// TIA Portal V20 export
DATA_BLOCK "CallEquipmentMotionCycle_DB"   // DB191
// stored: AssignedProDiagFB Unit1.Em1.ProDiag, InstanceOfName Unit1.Em1.CallEquipmentMotionCycle, InstanceOfType FB, Namespace Unit1.Em1
"Unit1.Em1.CallEquipmentMotionCycle"
   // VAR_INPUT
   //    diameter : LReal := 0.0;
   //    dancer : LReal := 0.105758101851848;
   // END_VAR
   // VAR_OUTPUT
   //    error { ExternalAccessible := 'False'; ExternalVisible := 'False'; ExternalWritable := 'False'} : Bool := FALSE;
   // END_VAR
   // VAR_IN_OUT
   //    syncNode : "Unit1.Em1.typeSyncNode";
   //    axis : Array[1.._.U1EM1_NO_OF_AXES] of DB_ANY;
   // END_VAR
   // VAR
   //    instSequenceUnwinderCycle : "Unit1.Em1.SequenceUnwinderCycle";
   // END_VAR
BEGIN
   instSequenceUnwinderCycle.enableHpMotion := FALSE;
   instSequenceUnwinderCycle.diameter := 0.0;
   instSequenceUnwinderCycle.dancer := 0.105758101851848;
   instSequenceUnwinderCycle.busy := FALSE;
   instSequenceUnwinderCycle.error := FALSE;
   instSequenceUnwinderCycle.slave := 141;
   instSequenceUnwinderCycle.master := 85;
   instSequenceUnwinderCycle.statFirstCall := FALSE;
   instSequenceUnwinderCycle.statDiameter := 0.0;
   instSequenceUnwinderCycle.statFrictionMeasurement.in.execute := FALSE;
   instSequenceUnwinderCycle.statFrictionMeasurement.in.abort := FALSE;
   instSequenceUnwinderCycle.statFrictionMeasurement.in.warmUpTime := T#30S;
   instSequenceUnwinderCycle.statFrictionMeasurement.in.rampTime := 1000.0;
   instSequenceUnwinderCycle.statFrictionMeasurement.in.noOfMeasurementPoints := 100;
   instSequenceUnwinderCycle.statFrictionMeasurement.in.sizeOfArray := 10;
   instSequenceUnwinderCycle.statFrictionMeasurement.in.maxSpeed := 0.0;
   instSequenceUnwinderCycle.statFrictionMeasurement.in.speedValues.values[0] := 100.0;
   instSequenceUnwinderCycle.statFrictionMeasurement.in.speedValues.values[1] := 200.0;
   instSequenceUnwinderCycle.statFrictionMeasurement.in.speedValues.values[2] := 300.0;
   instSequenceUnwinderCycle.statFrictionMeasurement.in.speedValues.values[3] := 400.0;
   instSequenceUnwinderCycle.statFrictionMeasurement.in.speedValues.values[4] := 500.0;
   instSequenceUnwinderCycle.statFrictionMeasurement.in.speedValues.values[5] := 600.0;
   instSequenceUnwinderCycle.statFrictionMeasurement.in.speedValues.values[6] := 700.0;
   instSequenceUnwinderCycle.statFrictionMeasurement.in.speedValues.values[7] := 800.0;
   instSequenceUnwinderCycle.statFrictionMeasurement.in.speedValues.values[8] := 900.0;
   instSequenceUnwinderCycle.statFrictionMeasurement.in.speedValues.values[9] := 1000.0;
   instSequenceUnwinderCycle.statFrictionMeasurement.in.speedValues.values[10..19] := 0.0;
   instSequenceUnwinderCycle.statFrictionMeasurement.in.measurementDelayTime := T#1S;
   instSequenceUnwinderCycle.statFrictionMeasurement.out.done := FALSE;
   instSequenceUnwinderCycle.statFrictionMeasurement.out.valid := FALSE;
   instSequenceUnwinderCycle.statFrictionMeasurement.out.aborted := FALSE;
   instSequenceUnwinderCycle.statFrictionMeasurement.out.busy := FALSE;
   instSequenceUnwinderCycle.statFrictionMeasurement.out.error := FALSE;
   instSequenceUnwinderCycle.statFrictionMeasurement.out.subfunctionState := 16#0000;
   instSequenceUnwinderCycle.statFrictionMeasurement.out.status := 16#7000;
   instSequenceUnwinderCycle.statMaxAcceleration := 360000.0;
   instSequenceUnwinderCycle.statMaxDeceleration := 360000.0;
   instSequenceUnwinderCycle.statUnitsLengthUnit := 1013;
   instSequenceUnwinderCycle.statUnitsVelocityUnit := 1062;
   instSequenceUnwinderCycle.statMechanicsLeadScrew := 10.0;
   instSequenceUnwinderCycle.statLengthConversion := 0.001;
   instSequenceUnwinderCycle.statVelocityConversion := 0.06;
   instSequenceUnwinderCycle.statAccelerationConversion := 0.001;
   instSequenceUnwinderCycle.instLConSMC_Winder.enable := FALSE;
   instSequenceUnwinderCycle.instLConSMC_Winder.speedMatch := FALSE;
   instSequenceUnwinderCycle.instLConSMC_Winder.cntrlEnable := FALSE;
   instSequenceUnwinderCycle.instLConSMC_Winder.jogPos := FALSE;
   instSequenceUnwinderCycle.instLConSMC_Winder.jogNeg := FALSE;
   instSequenceUnwinderCycle.instLConSMC_Winder.lineAxisMotionVector.s := 0.0;
   instSequenceUnwinderCycle.instLConSMC_Winder.lineAxisMotionVector.v := 0.0;
   instSequenceUnwinderCycle.instLConSMC_Winder.lineAxisMotionVector."a" := 0.0;
   instSequenceUnwinderCycle.instLConSMC_Winder.lineAxisActualValues.s := 0.0;
   instSequenceUnwinderCycle.instLConSMC_Winder.lineAxisActualValues.v := 0.0;
   instSequenceUnwinderCycle.instLConSMC_Winder.additionalVelocity := 0.0;
   instSequenceUnwinderCycle.instLConSMC_Winder.typeOfWinder := 2;
   instSequenceUnwinderCycle.instLConSMC_Winder.controlMode := 0;
   instSequenceUnwinderCycle.instLConSMC_Winder.typeOfDiameterCalc := 3;
   instSequenceUnwinderCycle.instLConSMC_Winder.holdDiameter := FALSE;
   instSequenceUnwinderCycle.instLConSMC_Winder.setDiameter := FALSE;
   instSequenceUnwinderCycle.instLConSMC_Winder.CntrlSetpoint := 0.0;
   instSequenceUnwinderCycle.instLConSMC_Winder.CntrlActual := 0.105758101851848;
   instSequenceUnwinderCycle.instLConSMC_Winder.tCycle := 10.0;
   instSequenceUnwinderCycle.instLConSMC_Winder.busy := FALSE;
   instSequenceUnwinderCycle.instLConSMC_Winder.active := FALSE;
   instSequenceUnwinderCycle.instLConSMC_Winder.ctrlBusy := FALSE;
   instSequenceUnwinderCycle.instLConSMC_Winder.inSync := FALSE;
   instSequenceUnwinderCycle.instLConSMC_Winder.error := FALSE;
   instSequenceUnwinderCycle.instLConSMC_Winder.errorID := 16#0000_0000;
   instSequenceUnwinderCycle.instLConSMC_Winder.winderAxis := 141;
   instSequenceUnwinderCycle.instLConSMC_Winder.diameter := 0.0;
   instSequenceUnwinderCycle.instLConSMC_Winder.statActive := FALSE;
   instSequenceUnwinderCycle.instLConSMC_Winder.statTel750Active := FALSE;
   instSequenceUnwinderCycle.instLConSMC_Winder.statEnableWebBreakDetection := FALSE;
   instSequenceUnwinderCycle.instLConSMC_Winder.statEnableWebBreakDetectionOld := FALSE;
   instSequenceUnwinderCycle.instLConSMC_Winder.statDancerControl := FALSE;
   instSequenceUnwinderCycle.instLConSMC_Winder.statEnableOld := FALSE;
   instSequenceUnwinderCycle.instLConSMC_Winder.statTorqueLimitUpperActive := FALSE;
   instSequenceUnwinderCycle.instLConSMC_Winder.statTorqueLimitLowerActive := FALSE;
   instSequenceUnwinderCycle.instLConSMC_Winder.statStartupError := FALSE;
   instSequenceUnwinderCycle.instLConSMC_Winder.statWinderAxisCtrl := FALSE;
   instSequenceUnwinderCycle.instLConSMC_Winder.statError := FALSE;
   instSequenceUnwinderCycle.instLConSMC_Winder.statInSync := FALSE;
   instSequenceUnwinderCycle.instLConSMC_Winder.statCtrlBusyInternal := FALSE;
   instSequenceUnwinderCycle.instLConSMC_Winder.statJogWinder := FALSE;
   instSequenceUnwinderCycle.instLConSMC_Winder.statBusy := FALSE;
   instSequenceUnwinderCycle.instLConSMC_Winder.statDeactivateJogDyn := TRUE;
   instSequenceUnwinderCycle.instLConSMC_Winder.statDisableAdditiveTorque := FALSE;
   instSequenceUnwinderCycle.instLConSMC_Winder.statCtrlBusyInternalOld := FALSE;
   instSequenceUnwinderCycle.instLConSMC_Winder.statNumberOfSamplesInternal := 1;
   instSequenceUnwinderCycle.instLConSMC_Winder.statNumberOfSamplesOld := 1;
   instSequenceUnwinderCycle.instLConSMC_Winder.statVeloUnit := 0;
   instSequenceUnwinderCycle.instLConSMC_Winder.statTorqueUnit := 0;
   instSequenceUnwinderCycle.instLConSMC_Winder.statControlMode := 0;
   instSequenceUnwinderCycle.instLConSMC_Winder.statTypeOfWinder := 0;
   instSequenceUnwinderCycle.instLConSMC_Winder.statFLineSpeed := 0;
   instSequenceUnwinderCycle.instLConSMC_Winder.statFPIDTorque := 0;
   instSequenceUnwinderCycle.instLConSMC_Winder.statFPIDSpeed := 0;
   instSequenceUnwinderCycle.instLConSMC_Winder.statFOverride := 0;
   instSequenceUnwinderCycle.instLConSMC_Winder.statActualTorque := 0.0;
   instSequenceUnwinderCycle.instLConSMC_Winder.statWinderAxisIntoRPM := 0.0;
   instSequenceUnwinderCycle.instLConSMC_Winder.statVelocityLUPerMin := 0.0;
   instSequenceUnwinderCycle.instLConSMC_Winder.statWndrTotalTorque := 0.0;
   instSequenceUnwinderCycle.instLConSMC_Winder.statTensionSpeedLUPerMin := 0.0;
   instSequenceUnwinderCycle.instLConSMC_Winder.statVelocitySetpointOld := 0.0;
   instSequenceUnwinderCycle.instLConSMC_Winder.statActShaftSpeed1PerMin := 0.0;
   instSequenceUnwinderCycle.instLConSMC_Winder.statIntDiameter := 0.31831;
   instSequenceUnwinderCycle.instLConSMC_Winder.statCircumference := 1.00000014952;
   instSequenceUnwinderCycle.instLConSMC_Winder.statTensionSetpoint := 0.0;
   instSequenceUnwinderCycle.instLConSMC_Winder.statDiameterPosition := 0.0;
   instSequenceUnwinderCycle.instLConSMC_Winder.statUpperTorqueLimitTOUnit := 0.0;
   instSequenceUnwinderCycle.instLConSMC_Winder.statLineVelocityInternalLUPerMin := 0.0;
   instSequenceUnwinderCycle.instLConSMC_Winder.statLineAccelerationInternalLUPerS2 := 0.0;
   instSequenceUnwinderCycle.instLConSMC_Winder.statDiameterVelocity := 0.0;
   instSequenceUnwinderCycle.instLConSMC_Winder.statLowerTorqueLimitTOUnit := 0.0;
   instSequenceUnwinderCycle.instLConSMC_Winder.statActDriveSpeed1PerMin := 0.0;
   instSequenceUnwinderCycle.instLConSMC_Winder.statSetDriveSpeed1PerMin := 0.0;
   instSequenceUnwinderCycle.instLConSMC_Winder.statSetShaftSpeed1PerMin := 0.0;
   instSequenceUnwinderCycle.instLConSMC_Winder.statWindingShaftSpeedSetpointPreCtrl1PerMin := 0.0;
   instSequenceUnwinderCycle.instLConSMC_Winder.statActSpeedOverride1PerMin := 16#FFF8_0000_0000_0000;
   instSequenceUnwinderCycle.instLConSMC_Winder.statReferenceTorque := 0.0;
   instSequenceUnwinderCycle.instLConSMC_Winder.statUpperTorqueLimitLimited := 0.0;
   instSequenceUnwinderCycle.instLConSMC_Winder.statLowerTorqueLimiLimited := 0.0;
   instSequenceUnwinderCycle.instLConSMC_Winder.statGearRatioInternal := 1.0;
   instSequenceUnwinderCycle.instLConSMC_Winder.statConvTorqueUnitToTO := 0.0;
   instSequenceUnwinderCycle.instLConSMC_Winder.statAddPos := 0.0;
   instSequenceUnwinderCycle.instLConSMC_Winder.statCommandMoveVelocityTOUnit := 0.0;
   instSequenceUnwinderCycle.instLConSMC_Winder.statReferenceVelocityTOUnit := 16#7FF0_0000_0000_0000;
   instSequenceUnwinderCycle.instLConSMC_Winder.statVDiff := 0.0;
   instSequenceUnwinderCycle.instLConSMC_Winder.statVsync := 0.0;
   instSequenceUnwinderCycle.instLConSMC_Winder.statOverride := 100.0;
   instSequenceUnwinderCycle.instLConSMC_Winder.statShaftFeedback := 195.934;
   instSequenceUnwinderCycle.instLConSMC_Winder.statPIDActualValue := 0.105758101851848;
   instSequenceUnwinderCycle.instLConSMC_Winder.statAxisDefaultAcc := 0.0;
   instSequenceUnwinderCycle.instLConSMC_Winder.statAxisDefaultJerk := 0.0;
   instSequenceUnwinderCycle.instLConSMC_Winder.statGearInternal.numerator := 1;
   instSequenceUnwinderCycle.instLConSMC_Winder.statGearInternal.denominator := 1;
   instSequenceUnwinderCycle.instLConSMC_Winder.statWinderMV.s := 0.0;
   instSequenceUnwinderCycle.instLConSMC_Winder.statWinderMV.v := 16#FFF8_0000_0000_0000;
   instSequenceUnwinderCycle.instLConSMC_Winder.statWinderMV."a" := 360.0;
   instSequenceUnwinderCycle.instLConSMC_Winder.statWinderMV.d := 360.0;
   instSequenceUnwinderCycle.instLConSMC_Winder.statWinderMV.j := 0.0;
   instSequenceUnwinderCycle.instLConSMC_Winder.statTorqueValues.upperTorqueLimit := 0.0;
   instSequenceUnwinderCycle.instLConSMC_Winder.statTorqueValues.lowerTorqueLimit := 0.0;
   instSequenceUnwinderCycle.instLConSMC_Winder.statTorqueValues.additiveTorque := 0.0;
   instSequenceUnwinderCycle.instLConSMC_Winder.statDynamicsInternalTOUnit.acceleration := 360.0;
   instSequenceUnwinderCycle.instLConSMC_Winder.statDynamicsInternalTOUnit.deceleration := 360.0;
   instSequenceUnwinderCycle.instLConSMC_Winder.statDynamicsInternalTOUnit.jerk := 0.0;
   instSequenceUnwinderCycle.instLConSMC_Winder.statDynamicsInternalTOUnit.abortAcceleration := TRUE;
   instSequenceUnwinderCycle.instLConSMC_Winder.instEnableInterface.enable := FALSE;
   instSequenceUnwinderCycle.instLConSMC_Winder.instEnableInterface.enableVelocityInterface := FALSE;
   instSequenceUnwinderCycle.instLConSMC_Winder.instEnableInterface.writeTorqueLimit := FALSE;
   instSequenceUnwinderCycle.instLConSMC_Winder.instEnableInterface.writeAdditiveTorque := FALSE;
   instSequenceUnwinderCycle.instLConSMC_Winder.instEnableInterface.positionControlled := FALSE;
   instSequenceUnwinderCycle.instLConSMC_Winder.instEnableInterface.referenceVelocity := 0.0;
   instSequenceUnwinderCycle.instLConSMC_Winder.instEnableInterface.override := 100.0;
   instSequenceUnwinderCycle.instLConSMC_Winder.instEnableInterface.valid := FALSE;
   instSequenceUnwinderCycle.instLConSMC_Winder.instEnableInterface.busy := FALSE;
   instSequenceUnwinderCycle.instLConSMC_Winder.instEnableInterface.error := FALSE;
   instSequenceUnwinderCycle.instLConSMC_Winder.instEnableInterface.status := 16#0000_7000;
   instSequenceUnwinderCycle.instLConSMC_Winder.instEnableInterface.subfunctionState := 16#0000;
   instSequenceUnwinderCycle.instLConSMC_Winder.instEnableInterface.MCInterfaceActive := FALSE;
   instSequenceUnwinderCycle.instLConSMC_Winder.instEnableInterface.additiveTorqueActive := FALSE;
   instSequenceUnwinderCycle.instLConSMC_Winder.instEnableInterface.torqueLimitActive := FALSE;
   instSequenceUnwinderCycle.instLConSMC_Winder.instEnableInterface.axis := 141;
   instSequenceUnwinderCycle.instLConSMC_Winder.instEnableInterface.statEnableOld := FALSE;
   instSequenceUnwinderCycle.instLConSMC_Winder.instEnableInterface.statValid := FALSE;
   instSequenceUnwinderCycle.instLConSMC_Winder.instEnableInterface.statBusy := FALSE;
   instSequenceUnwinderCycle.instLConSMC_Winder.instEnableInterface.statError := FALSE;
   instSequenceUnwinderCycle.instLConSMC_Winder.instEnableInterface.statErrorUserCleared := FALSE;
   instSequenceUnwinderCycle.instLConSMC_Winder.instEnableInterface.statErrorAutoCleared := FALSE;
   instSequenceUnwinderCycle.instLConSMC_Winder.instEnableInterface.statAdditiveTorqueActive := FALSE;
   instSequenceUnwinderCycle.instLConSMC_Winder.instEnableInterface.statDisablingCompleted := FALSE;
   instSequenceUnwinderCycle.instLConSMC_Winder.instEnableInterface.statTorqueLimitActive := FALSE;
   instSequenceUnwinderCycle.instLConSMC_Winder.instEnableInterface.statMCInterfaceActive := FALSE;
   instSequenceUnwinderCycle.instLConSMC_Winder.instEnableInterface.statEnableAdditiveTorque := FALSE;
   instSequenceUnwinderCycle.instLConSMC_Winder.instEnableInterface.statEnableTorqueLimit := FALSE;
   instSequenceUnwinderCycle.instLConSMC_Winder.instEnableInterface.statExecuteMoveVelocity := FALSE;
   instSequenceUnwinderCycle.instLConSMC_Winder.instEnableInterface.statExecuteStop := FALSE;
   instSequenceUnwinderCycle.instLConSMC_Winder.instEnableInterface.statInternalMoveExecute := FALSE;
   instSequenceUnwinderCycle.instLConSMC_Winder.instEnableInterface.statRefTOValid := FALSE;
   instSequenceUnwinderCycle.instLConSMC_Winder.instEnableInterface.statFirstStepCycle := FALSE;
   instSequenceUnwinderCycle.instLConSMC_Winder.instEnableInterface.statDecelerationOld := 0.0;
   instSequenceUnwinderCycle.instLConSMC_Winder.instEnableInterface.statAccelerationOld := 0.0;
   instSequenceUnwinderCycle.instLConSMC_Winder.instEnableInterface.statJerkOld := 0.0;
   instSequenceUnwinderCycle.instLConSMC_Winder.instEnableInterface.statReferenceVelocityOld := 0.0;
   instSequenceUnwinderCycle.instLConSMC_Winder.instEnableInterface.statAxisInt := 0;
   instSequenceUnwinderCycle.instLConSMC_Winder.instEnableInterface.instStop.Execute := FALSE;
   instSequenceUnwinderCycle.instLConSMC_Winder.instEnableInterface.instStop.Deceleration := -1.0;
   instSequenceUnwinderCycle.instLConSMC_Winder.instEnableInterface.instStop.Jerk := -1.0;
   instSequenceUnwinderCycle.instLConSMC_Winder.instEnableInterface.instStop.AbortAcceleration := FALSE;
   instSequenceUnwinderCycle.instLConSMC_Winder.instEnableInterface.instStop.Mode := 0;
   instSequenceUnwinderCycle.instLConSMC_Winder.instEnableInterface.instStop.Done := FALSE;
   instSequenceUnwinderCycle.instLConSMC_Winder.instEnableInterface.instStop.Busy := FALSE;
   instSequenceUnwinderCycle.instLConSMC_Winder.instEnableInterface.instStop.CommandAborted := FALSE;
   instSequenceUnwinderCycle.instLConSMC_Winder.instEnableInterface.instStop.Error := FALSE;
   instSequenceUnwinderCycle.instLConSMC_Winder.instEnableInterface.instStop.ErrorId := 16#0000;
   instSequenceUnwinderCycle.instLConSMC_Winder.instEnableInterface.instMoveVelocity.Execute := FALSE;
   instSequenceUnwinderCycle.instLConSMC_Winder.instEnableInterface.instMoveVelocity.Velocity := 100.0;
   instSequenceUnwinderCycle.instLConSMC_Winder.instEnableInterface.instMoveVelocity.Acceleration := -1.0;
   instSequenceUnwinderCycle.instLConSMC_Winder.instEnableInterface.instMoveVelocity.Deceleration := -1.0;
   instSequenceUnwinderCycle.instLConSMC_Winder.instEnableInterface.instMoveVelocity.Jerk := -1.0;
   instSequenceUnwinderCycle.instLConSMC_Winder.instEnableInterface.instMoveVelocity.Direction := 0;
   instSequenceUnwinderCycle.instLConSMC_Winder.instEnableInterface.instMoveVelocity.Current := FALSE;
   instSequenceUnwinderCycle.instLConSMC_Winder.instEnableInterface.instMoveVelocity.PositionControlled := TRUE;
   instSequenceUnwinderCycle.instLConSMC_Winder.instEnableInterface.instMoveVelocity.InVelocity := FALSE;
   instSequenceUnwinderCycle.instLConSMC_Winder.instEnableInterface.instMoveVelocity.Busy := FALSE;
   instSequenceUnwinderCycle.instLConSMC_Winder.instEnableInterface.instMoveVelocity.CommandAborted := FALSE;
   instSequenceUnwinderCycle.instLConSMC_Winder.instEnableInterface.instMoveVelocity.Error := FALSE;
   instSequenceUnwinderCycle.instLConSMC_Winder.instEnableInterface.instMoveVelocity.ErrorId := 16#0000;
   instSequenceUnwinderCycle.instLConSMC_Winder.instEnableInterface.instTorqueAdditive.Enable := FALSE;
   instSequenceUnwinderCycle.instLConSMC_Winder.instEnableInterface.instTorqueAdditive.Value := 0.0;
   instSequenceUnwinderCycle.instLConSMC_Winder.instEnableInterface.instTorqueAdditive.Busy := FALSE;
   instSequenceUnwinderCycle.instLConSMC_Winder.instEnableInterface.instTorqueAdditive.Error := FALSE;
   instSequenceUnwinderCycle.instLConSMC_Winder.instEnableInterface.instTorqueAdditive.ErrorId := 16#0000;
   instSequenceUnwinderCycle.instLConSMC_Winder.instEnableInterface.instTorqueRange.Enable := FALSE;
   instSequenceUnwinderCycle.instLConSMC_Winder.instEnableInterface.instTorqueRange.UpperLimit := 1000000000000.0;
   instSequenceUnwinderCycle.instLConSMC_Winder.instEnableInterface.instTorqueRange.LowerLimit := -1000000000000.0;
   instSequenceUnwinderCycle.instLConSMC_Winder.instEnableInterface.instTorqueRange.Busy := FALSE;
   instSequenceUnwinderCycle.instLConSMC_Winder.instEnableInterface.instTorqueRange.Error := FALSE;
   instSequenceUnwinderCycle.instLConSMC_Winder.instEnableInterface.instTorqueRange.ErrorId := 16#0000;
   instSequenceUnwinderCycle.instLConSMC_Winder.instEnableInterface.instRTrigEnableInterface.CLK := FALSE;
   instSequenceUnwinderCycle.instLConSMC_Winder.instEnableInterface.instRTrigEnableInterface.Q := FALSE;
   instSequenceUnwinderCycle.instLConSMC_Winder.instEnableInterface.instRTrigEnableInterface.Stat_Bit := FALSE;
   instSequenceUnwinderCycle.instLConSMC_Winder.instEnableInterface.statSubfunctionState := 16#0000;
   instSequenceUnwinderCycle.instLConSMC_Winder.instEnableInterface.statStatus := 16#0000_7000;
   instSequenceUnwinderCycle.instLConSMC_Winder.instEnableInterface.statFBState := 0;
   instSequenceUnwinderCycle.instLConSMC_Winder.instEnableInterface.statFBStateOld := 0;
   instSequenceUnwinderCycle.instLConSMC_Winder.instTPID.enable := FALSE;
   instSequenceUnwinderCycle.instLConSMC_Winder.instTPID.openLoopCtrl := FALSE;
   instSequenceUnwinderCycle.instLConSMC_Winder.instTPID.setpointValue := 0.0;
   instSequenceUnwinderCycle.instLConSMC_Winder.instTPID.actualValue := 0.105758101851848;
   instSequenceUnwinderCycle.instLConSMC_Winder.instTPID.preControl := 0.0;
   instSequenceUnwinderCycle.instLConSMC_Winder.instTPID.adaptionValue := 0.0;
   instSequenceUnwinderCycle.instLConSMC_Winder.instTPID.holdIntChannel := FALSE;
   instSequenceUnwinderCycle.instLConSMC_Winder.instTPID.setIntChannel := FALSE;
   instSequenceUnwinderCycle.instLConSMC_Winder.instTPID.x1 := 0.0;
   instSequenceUnwinderCycle.instLConSMC_Winder.instTPID.Kp1 := 10.0;
   instSequenceUnwinderCycle.instLConSMC_Winder.instTPID.x2 := 0.0;
   instSequenceUnwinderCycle.instLConSMC_Winder.instTPID.Kp2 := 0.0;
   instSequenceUnwinderCycle.instLConSMC_Winder.instTPID.limRampTime := 300.0;
   instSequenceUnwinderCycle.instLConSMC_Winder.instTPID.setNominalValue := 100.0;
   instSequenceUnwinderCycle.instLConSMC_Winder.instTPID.setRampTime := 500.0;
   instSequenceUnwinderCycle.instLConSMC_Winder.instTPID.integTime := 200.0;
   instSequenceUnwinderCycle.instLConSMC_Winder.instTPID.derivTime := 0.0;
   instSequenceUnwinderCycle.instLConSMC_Winder.instTPID.filterTime := 10.0;
   instSequenceUnwinderCycle.instLConSMC_Winder.instTPID.intSetValue := 0.0;
   instSequenceUnwinderCycle.instLConSMC_Winder.instTPID.controlMode := FALSE;
   instSequenceUnwinderCycle.instLConSMC_Winder.instTPID.deadBand := 0.0;
   instSequenceUnwinderCycle.instLConSMC_Winder.instTPID.outValueFactor := -1.0;
   instSequenceUnwinderCycle.instLConSMC_Winder.instTPID.upperLimit := 2.0;
   instSequenceUnwinderCycle.instLConSMC_Winder.instTPID.lowerLimit := -5.0;
   instSequenceUnwinderCycle.instLConSMC_Winder.instTPID.tCycle := 10.0;
   instSequenceUnwinderCycle.instLConSMC_Winder.instTPID.busy := FALSE;
   instSequenceUnwinderCycle.instLConSMC_Winder.instTPID.error := FALSE;
   instSequenceUnwinderCycle.instLConSMC_Winder.instTPID.errorId := 16#0000_0000;
   instSequenceUnwinderCycle.instLConSMC_Winder.instTPID.upperLimReached := FALSE;
   instSequenceUnwinderCycle.instLConSMC_Winder.instTPID.lowerLimReached := FALSE;
   instSequenceUnwinderCycle.instLConSMC_Winder.instTPID.RFGLimReached := FALSE;
   instSequenceUnwinderCycle.instLConSMC_Winder.instTPID.RFGSetpointReached := FALSE;
   instSequenceUnwinderCycle.instLConSMC_Winder.instTPID.RFGSetpointValue := 0.0;
   instSequenceUnwinderCycle.instLConSMC_Winder.instTPID.outValue := 0.0;
   instSequenceUnwinderCycle.instLConSMC_Winder.instTPID.effectiveKp := 0.0;
   instSequenceUnwinderCycle.instLConSMC_Winder.instTPID.statEnableOld := FALSE;
   instSequenceUnwinderCycle.instLConSMC_Winder.instTPID.instRFGLim.x := 0.0;
   instSequenceUnwinderCycle.instLConSMC_Winder.instTPID.instRFGLim.nominalValue := 1.0;
   instSequenceUnwinderCycle.instLConSMC_Winder.instTPID.instRFGLim.upperLimit := 0.0;
   instSequenceUnwinderCycle.instLConSMC_Winder.instTPID.instRFGLim.lowerLimit := 0.0;
   instSequenceUnwinderCycle.instLConSMC_Winder.instTPID.instRFGLim.setValue := 0.0;
   instSequenceUnwinderCycle.instLConSMC_Winder.instTPID.instRFGLim.rampupTime := 0.0;
   instSequenceUnwinderCycle.instLConSMC_Winder.instTPID.instRFGLim.rampdownTime := 0.0;
   instSequenceUnwinderCycle.instLConSMC_Winder.instTPID.instRFGLim.rampTimeMode := 0;
   instSequenceUnwinderCycle.instLConSMC_Winder.instTPID.instRFGLim.set := FALSE;
   instSequenceUnwinderCycle.instLConSMC_Winder.instTPID.instRFGLim.followup := FALSE;
   instSequenceUnwinderCycle.instLConSMC_Winder.instTPID.instRFGLim.increase := FALSE;
   instSequenceUnwinderCycle.instLConSMC_Winder.instTPID.instRFGLim.decrease := FALSE;
   instSequenceUnwinderCycle.instLConSMC_Winder.instTPID.instRFGLim.tCycle := 0.0;
   instSequenceUnwinderCycle.instLConSMC_Winder.instTPID.instRFGLim.error := FALSE;
   instSequenceUnwinderCycle.instLConSMC_Winder.instTPID.instRFGLim.errorID := 16#0000_0000;
   instSequenceUnwinderCycle.instLConSMC_Winder.instTPID.instRFGLim.y := 0.0;
   instSequenceUnwinderCycle.instLConSMC_Winder.instTPID.instRFGLim.ya := 0.0;
   instSequenceUnwinderCycle.instLConSMC_Winder.instTPID.instRFGLim.SetpointReached := FALSE;
   instSequenceUnwinderCycle.instLConSMC_Winder.instTPID.instRFGLim.upperLimitReached := FALSE;
   instSequenceUnwinderCycle.instLConSMC_Winder.instTPID.instRFGLim.lowerLimitReached := FALSE;
   instSequenceUnwinderCycle.instLConSMC_Winder.instTPID.instRFGLim.statTUs := 0.0;
   instSequenceUnwinderCycle.instLConSMC_Winder.instTPID.instRFGLim.statTDs := 0.0;
   instSequenceUnwinderCycle.instLConSMC_Winder.instTPID.instRFGLim.statYkm1 := 0.0;
   instSequenceUnwinderCycle.instLConSMC_Winder.instTPID.instRFGLim.statLLs := 0.0;
   instSequenceUnwinderCycle.instLConSMC_Winder.instTPID.instRFGLim.statXs := 0.0;
   instSequenceUnwinderCycle.instLConSMC_Winder.instTPID.instRFGLim.stat1 := 0.0;
   instSequenceUnwinderCycle.instLConSMC_Winder.instTPID.instRFGLim.statError := FALSE;
   instSequenceUnwinderCycle.instLConSMC_Winder.instTPID.instRFGLim.statY := 0.0;
   instSequenceUnwinderCycle.instLConSMC_Winder.instTPID.instRFGSet.x := 0.0;
   instSequenceUnwinderCycle.instLConSMC_Winder.instTPID.instRFGSet.nominalValue := 1.0;
   instSequenceUnwinderCycle.instLConSMC_Winder.instTPID.instRFGSet.upperLimit := 0.0;
   instSequenceUnwinderCycle.instLConSMC_Winder.instTPID.instRFGSet.lowerLimit := 0.0;
   instSequenceUnwinderCycle.instLConSMC_Winder.instTPID.instRFGSet.setValue := 0.0;
   instSequenceUnwinderCycle.instLConSMC_Winder.instTPID.instRFGSet.rampupTime := 0.0;
   instSequenceUnwinderCycle.instLConSMC_Winder.instTPID.instRFGSet.rampdownTime := 0.0;
   instSequenceUnwinderCycle.instLConSMC_Winder.instTPID.instRFGSet.rampTimeMode := 0;
   instSequenceUnwinderCycle.instLConSMC_Winder.instTPID.instRFGSet.set := FALSE;
   instSequenceUnwinderCycle.instLConSMC_Winder.instTPID.instRFGSet.followup := FALSE;
   instSequenceUnwinderCycle.instLConSMC_Winder.instTPID.instRFGSet.increase := FALSE;
   instSequenceUnwinderCycle.instLConSMC_Winder.instTPID.instRFGSet.decrease := FALSE;
   instSequenceUnwinderCycle.instLConSMC_Winder.instTPID.instRFGSet.tCycle := 0.0;
   instSequenceUnwinderCycle.instLConSMC_Winder.instTPID.instRFGSet.error := FALSE;
   instSequenceUnwinderCycle.instLConSMC_Winder.instTPID.instRFGSet.errorID := 16#0000_0000;
   instSequenceUnwinderCycle.instLConSMC_Winder.instTPID.instRFGSet.y := 0.0;
   instSequenceUnwinderCycle.instLConSMC_Winder.instTPID.instRFGSet.ya := 0.0;
   instSequenceUnwinderCycle.instLConSMC_Winder.instTPID.instRFGSet.SetpointReached := FALSE;
   instSequenceUnwinderCycle.instLConSMC_Winder.instTPID.instRFGSet.upperLimitReached := FALSE;
   instSequenceUnwinderCycle.instLConSMC_Winder.instTPID.instRFGSet.lowerLimitReached := FALSE;
   instSequenceUnwinderCycle.instLConSMC_Winder.instTPID.instRFGSet.statTUs := 0.0;
   instSequenceUnwinderCycle.instLConSMC_Winder.instTPID.instRFGSet.statTDs := 0.0;
   instSequenceUnwinderCycle.instLConSMC_Winder.instTPID.instRFGSet.statYkm1 := 0.0;
   instSequenceUnwinderCycle.instLConSMC_Winder.instTPID.instRFGSet.statLLs := 0.0;
   instSequenceUnwinderCycle.instLConSMC_Winder.instTPID.instRFGSet.statXs := 0.0;
   instSequenceUnwinderCycle.instLConSMC_Winder.instTPID.instRFGSet.stat1 := 0.0;
   instSequenceUnwinderCycle.instLConSMC_Winder.instTPID.instRFGSet.statError := FALSE;
   instSequenceUnwinderCycle.instLConSMC_Winder.instTPID.instRFGSet.statY := 0.0;
   instSequenceUnwinderCycle.instLConSMC_Winder.instTPID.instPidController.enable := TRUE;
   instSequenceUnwinderCycle.instLConSMC_Winder.instTPID.instPidController.reset := TRUE;
   instSequenceUnwinderCycle.instLConSMC_Winder.instTPID.instPidController.setpointValue := 0.0;
   instSequenceUnwinderCycle.instLConSMC_Winder.instTPID.instPidController.actualValue := 0.105758101851848;
   instSequenceUnwinderCycle.instLConSMC_Winder.instTPID.instPidController.preControl := 0.0;
   instSequenceUnwinderCycle.instLConSMC_Winder.instTPID.instPidController.propGain := 0.0;
   instSequenceUnwinderCycle.instLConSMC_Winder.instTPID.instPidController.integTime := 200.0;
   instSequenceUnwinderCycle.instLConSMC_Winder.instTPID.instPidController.derivTime := 0.0;
   instSequenceUnwinderCycle.instLConSMC_Winder.instTPID.instPidController.filterTime := 10.0;
   instSequenceUnwinderCycle.instLConSMC_Winder.instTPID.instPidController.upperLimit := 0.0;
   instSequenceUnwinderCycle.instLConSMC_Winder.instTPID.instPidController.lowerLimit := 0.0;
   instSequenceUnwinderCycle.instLConSMC_Winder.instTPID.instPidController.intSetValue := 0.0;
   instSequenceUnwinderCycle.instLConSMC_Winder.instTPID.instPidController.holdIntChannel := FALSE;
   instSequenceUnwinderCycle.instLConSMC_Winder.instTPID.instPidController.setIntChannel := FALSE;
   instSequenceUnwinderCycle.instLConSMC_Winder.instTPID.instPidController.controlMode := FALSE;
   instSequenceUnwinderCycle.instLConSMC_Winder.instTPID.instPidController.deadBand := 0.0;
   instSequenceUnwinderCycle.instLConSMC_Winder.instTPID.instPidController.actualValueFactor := 1.0;
   instSequenceUnwinderCycle.instLConSMC_Winder.instTPID.instPidController.actualValueOffset := 0.0;
   instSequenceUnwinderCycle.instLConSMC_Winder.instTPID.instPidController.outValueFactor := -1.0;
   instSequenceUnwinderCycle.instLConSMC_Winder.instTPID.instPidController.outValueOffset := 0.0;
   instSequenceUnwinderCycle.instLConSMC_Winder.instTPID.instPidController.tCycle := 10.0;
   instSequenceUnwinderCycle.instLConSMC_Winder.instTPID.instPidController.busy := TRUE;
   instSequenceUnwinderCycle.instLConSMC_Winder.instTPID.instPidController.error := FALSE;
   instSequenceUnwinderCycle.instLConSMC_Winder.instTPID.instPidController.errorID := 16#0000_0000;
   instSequenceUnwinderCycle.instLConSMC_Winder.instTPID.instPidController.upperLimitReached := TRUE;
   instSequenceUnwinderCycle.instLConSMC_Winder.instTPID.instPidController.lowerLimitReached := TRUE;
   instSequenceUnwinderCycle.instLConSMC_Winder.instTPID.instPidController.deviationValue := -0.105758101851848;
   instSequenceUnwinderCycle.instLConSMC_Winder.instTPID.instPidController.pOutValue := 0.0;
   instSequenceUnwinderCycle.instLConSMC_Winder.instTPID.instPidController.iOutValue := 0.0;
   instSequenceUnwinderCycle.instLConSMC_Winder.instTPID.instPidController.dOutValue := 0.0;
   instSequenceUnwinderCycle.instLConSMC_Winder.instTPID.instPidController.outValue := 0.0;
   instSequenceUnwinderCycle.instLConSMC_Winder.instTPID.instPidController.statDeviationPrev := 0.0;
   instSequenceUnwinderCycle.instLConSMC_Winder.instTPID.instPidController.statActPT1Prev := 0.105758101851848;
   instSequenceUnwinderCycle.instLConSMC_Winder.instTPID.instPidController.statFirstRun := FALSE;
   instSequenceUnwinderCycle.instLConSMC_Winder.instTPID.instPidController.statError := FALSE;
   instSequenceUnwinderCycle.instLConSMC_Winder.instTPID.instPidController.statBusy := TRUE;
   instSequenceUnwinderCycle.instLConSMC_Winder.instTPID.instPidController.statUpperLimitReached := TRUE;
   instSequenceUnwinderCycle.instLConSMC_Winder.instTPID.instPidController.statLowerLimitReached := TRUE;
   instSequenceUnwinderCycle.instLConSMC_Winder.instTPID.instPidController.statErrorID := 16#0000_0000;
   instSequenceUnwinderCycle.instLConSMC_Winder.instTPID.instPidController.statDiff := 0.0;
   instSequenceUnwinderCycle.instLConSMC_Winder.instTPID.instPidController.statActualVal := 0.105758101851848;
   instSequenceUnwinderCycle.instLConSMC_Winder.instTPID.instPidController.statTi := 200.0;
   instSequenceUnwinderCycle.instLConSMC_Winder.instTPID.instPidController.statTd := 0.0;
   instSequenceUnwinderCycle.instLConSMC_Winder.instTPID.instPidController.statEnableOld := TRUE;
   instSequenceUnwinderCycle.instLConSMC_Winder.instTPID.instPidController.statY := 0.105758101851848;
   instSequenceUnwinderCycle.instLConSMC_Winder.instTPID.instPidController.statPOutValue := 0.0;
   instSequenceUnwinderCycle.instLConSMC_Winder.instTPID.instPidController.statIOutValue := 0.0;
   instSequenceUnwinderCycle.instLConSMC_Winder.instTPID.instPidController.statDOutValue := 0.0;
   instSequenceUnwinderCycle.instLConSMC_Winder.instTPID.instPidController.statOutValue := 0.0;
   instSequenceUnwinderCycle.instLConSMC_Winder.instTPID.instPidController.statDeviationValue := -0.105758101851848;
   instSequenceUnwinderCycle.instLConSMC_Winder.instTPID.instPidController.instPT1.set := TRUE;
   instSequenceUnwinderCycle.instLConSMC_Winder.instTPID.instPidController.instPT1.x := 0.105758101851848;
   instSequenceUnwinderCycle.instLConSMC_Winder.instTPID.instPidController.instPT1.setvalue := 0.105758101851848;
   instSequenceUnwinderCycle.instLConSMC_Winder.instTPID.instPidController.instPT1.smoothingTime := 10.0;
   instSequenceUnwinderCycle.instLConSMC_Winder.instTPID.instPidController.instPT1.tCycle := 10.0;
   instSequenceUnwinderCycle.instLConSMC_Winder.instTPID.instPidController.instPT1.error := FALSE;
   instSequenceUnwinderCycle.instLConSMC_Winder.instTPID.instPidController.instPT1.errorID := 16#0000_0000;
   instSequenceUnwinderCycle.instLConSMC_Winder.instTPID.instPidController.instPT1.y := 0.105758101851848;
   instSequenceUnwinderCycle.instLConSMC_Winder.instTPID.instPidController.instPT1.statTmax := 0.0;
   instSequenceUnwinderCycle.instLConSMC_Winder.instTPID.instPidController.instPT1.statXkm1 := 0.105758101851848;
   instSequenceUnwinderCycle.instLConSMC_Winder.instTPID.instPidController.instPT1.statYkm1 := 0.105758101851848;
   instSequenceUnwinderCycle.instLConSMC_Winder.instTPID.instPidController.instPT1.statFirstRun := FALSE;
   instSequenceUnwinderCycle.instLConSMC_Winder.instTPID.instPidController.instPT1.statY := 0.105758101851848;
   instSequenceUnwinderCycle.instLConSMC_Winder.instTPID.statEffSetPoint := 0.0;
   instSequenceUnwinderCycle.instLConSMC_Winder.instTPID.statEffLimit := 0.0;
   instSequenceUnwinderCycle.instLConSMC_Winder.instTPID.statLimRFGSetVal := 0.0;
   instSequenceUnwinderCycle.instLConSMC_Winder.instTPID.statOutValue := 0.0;
   instSequenceUnwinderCycle.instLConSMC_Winder.instTPID.statEffectiveKp := 0.0;
   instSequenceUnwinderCycle.instLConSMC_Winder.instTorquePrecontrol.enable := FALSE;
   instSequenceUnwinderCycle.instLConSMC_Winder.instTorquePrecontrol.torqueOn := FALSE;
   instSequenceUnwinderCycle.instLConSMC_Winder.instTorquePrecontrol.metricUnits := TRUE;
   instSequenceUnwinderCycle.instLConSMC_Winder.instTorquePrecontrol.typeOfWinder := 0;
   instSequenceUnwinderCycle.instLConSMC_Winder.instTorquePrecontrol.drivespeed := 0.0;
   instSequenceUnwinderCycle.instLConSMC_Winder.instTorquePrecontrol.lineSpeed := 0.0;
   instSequenceUnwinderCycle.instLConSMC_Winder.instTorquePrecontrol.lineAcceleration := 0.0;
   instSequenceUnwinderCycle.instLConSMC_Winder.instTorquePrecontrol.diamActVal := 0.0;
   instSequenceUnwinderCycle.instLConSMC_Winder.instTorquePrecontrol.tensionSetpoint := 0.0;
   instSequenceUnwinderCycle.instLConSMC_Winder.instTorquePrecontrol.additiveTorque := 0.0;
   instSequenceUnwinderCycle.instLConSMC_Winder.instTorquePrecontrol.density := 1000.0;
   instSequenceUnwinderCycle.instLConSMC_Winder.instTorquePrecontrol.diamMin := 0.075;
   instSequenceUnwinderCycle.instLConSMC_Winder.instTorquePrecontrol.diamMax := 0.6;
   instSequenceUnwinderCycle.instLConSMC_Winder.instTorquePrecontrol.width := 0.2;
   instSequenceUnwinderCycle.instLConSMC_Winder.instTorquePrecontrol.fillFactor := 1.0;
   instSequenceUnwinderCycle.instLConSMC_Winder.instTorquePrecontrol.JFix := 0.0;
   instSequenceUnwinderCycle.instLConSMC_Winder.instTorquePrecontrol.JMandrel := 0.0;
   instSequenceUnwinderCycle.instLConSMC_Winder.instTorquePrecontrol.JMot := 8.0E-05;
   instSequenceUnwinderCycle.instLConSMC_Winder.instTorquePrecontrol.gearRatio := 1.0;
   instSequenceUnwinderCycle.instLConSMC_Winder.instTorquePrecontrol.frictionAdjustment := 0.0;
   instSequenceUnwinderCycle.instLConSMC_Winder.instTorquePrecontrol.tensionAdjustment := 1.0;
   instSequenceUnwinderCycle.instLConSMC_Winder.instTorquePrecontrol.accelerationAdjustment := 0.0;
   instSequenceUnwinderCycle.instLConSMC_Winder.instTorquePrecontrol.dDdTAdjustment := 0.0;
   instSequenceUnwinderCycle.instLConSMC_Winder.instTorquePrecontrol.sizeOfArray := 10;
   instSequenceUnwinderCycle.instLConSMC_Winder.instTorquePrecontrol.xn_speedValues.values[0] := 300.0;
   instSequenceUnwinderCycle.instLConSMC_Winder.instTorquePrecontrol.xn_speedValues.values[1] := 600.0;
   instSequenceUnwinderCycle.instLConSMC_Winder.instTorquePrecontrol.xn_speedValues.values[2] := 900.0;
   instSequenceUnwinderCycle.instLConSMC_Winder.instTorquePrecontrol.xn_speedValues.values[3] := 1200.0;
   instSequenceUnwinderCycle.instLConSMC_Winder.instTorquePrecontrol.xn_speedValues.values[4] := 1500.0;
   instSequenceUnwinderCycle.instLConSMC_Winder.instTorquePrecontrol.xn_speedValues.values[5] := 1800.0;
   instSequenceUnwinderCycle.instLConSMC_Winder.instTorquePrecontrol.xn_speedValues.values[6] := 2100.0;
   instSequenceUnwinderCycle.instLConSMC_Winder.instTorquePrecontrol.xn_speedValues.values[7] := 2400.0;
   instSequenceUnwinderCycle.instLConSMC_Winder.instTorquePrecontrol.xn_speedValues.values[8] := 2700.0;
   instSequenceUnwinderCycle.instLConSMC_Winder.instTorquePrecontrol.xn_speedValues.values[9] := 3000.0;
   instSequenceUnwinderCycle.instLConSMC_Winder.instTorquePrecontrol.xn_speedValues.values[10..19] := 0.0;
   instSequenceUnwinderCycle.instLConSMC_Winder.instTorquePrecontrol.yn_torqueValues.values[0] := 0.3384;
   instSequenceUnwinderCycle.instLConSMC_Winder.instTorquePrecontrol.yn_torqueValues.values[1] := 0.4516;
   instSequenceUnwinderCycle.instLConSMC_Winder.instTorquePrecontrol.yn_torqueValues.values[2] := 0.5326;
   instSequenceUnwinderCycle.instLConSMC_Winder.instTorquePrecontrol.yn_torqueValues.values[3] := 0.6176;
   instSequenceUnwinderCycle.instLConSMC_Winder.instTorquePrecontrol.yn_torqueValues.values[4] := 0.7165;
   instSequenceUnwinderCycle.instLConSMC_Winder.instTorquePrecontrol.yn_torqueValues.values[5] := 0.8168;
   instSequenceUnwinderCycle.instLConSMC_Winder.instTorquePrecontrol.yn_torqueValues.values[6] := 0.9135;
   instSequenceUnwinderCycle.instLConSMC_Winder.instTorquePrecontrol.yn_torqueValues.values[7] := 0.9894;
   instSequenceUnwinderCycle.instLConSMC_Winder.instTorquePrecontrol.yn_torqueValues.values[8] := 1.0461;
   instSequenceUnwinderCycle.instLConSMC_Winder.instTorquePrecontrol.yn_torqueValues.values[9] := 1.1249;
   instSequenceUnwinderCycle.instLConSMC_Winder.instTorquePrecontrol.yn_torqueValues.values[10..19] := 0.0;
   instSequenceUnwinderCycle.instLConSMC_Winder.instTorquePrecontrol.tCycle := 10.0;
   instSequenceUnwinderCycle.instLConSMC_Winder.instTorquePrecontrol.busy := FALSE;
   instSequenceUnwinderCycle.instLConSMC_Winder.instTorquePrecontrol.error := FALSE;
   instSequenceUnwinderCycle.instLConSMC_Winder.instTorquePrecontrol.errorID := 16#0000_0000;
   instSequenceUnwinderCycle.instLConSMC_Winder.instTorquePrecontrol.totalinertia := 0.0;
   instSequenceUnwinderCycle.instLConSMC_Winder.instTorquePrecontrol.mass := 0.0;
   instSequenceUnwinderCycle.instLConSMC_Winder.instTorquePrecontrol.preCtrlMotor := 0.0;
   instSequenceUnwinderCycle.instLConSMC_Winder.instTorquePrecontrol.totalTorquePreCtrl := 0.0;
   instSequenceUnwinderCycle.instLConSMC_Winder.instTorquePrecontrol.variableInertia := 0.0;
   instSequenceUnwinderCycle.instLConSMC_Winder.instTorquePrecontrol.maxInertia := 0.0;
   instSequenceUnwinderCycle.instLConSMC_Winder.instTorquePrecontrol.tensionTorque := 0.0;
   instSequenceUnwinderCycle.instLConSMC_Winder.instTorquePrecontrol.instTableChar.enable := FALSE;
   instSequenceUnwinderCycle.instLConSMC_Winder.instTorquePrecontrol.instTableChar.x := 0.0;
   instSequenceUnwinderCycle.instLConSMC_Winder.instTorquePrecontrol.instTableChar.sizeOfArray := 20;
   instSequenceUnwinderCycle.instLConSMC_Winder.instTorquePrecontrol.instTableChar.xn.values[0..19] := 0.0;
   instSequenceUnwinderCycle.instLConSMC_Winder.instTorquePrecontrol.instTableChar.yn.values[0..19] := 0.0;
   instSequenceUnwinderCycle.instLConSMC_Winder.instTorquePrecontrol.instTableChar.busy := FALSE;
   instSequenceUnwinderCycle.instLConSMC_Winder.instTorquePrecontrol.instTableChar.error := FALSE;
   instSequenceUnwinderCycle.instLConSMC_Winder.instTorquePrecontrol.instTableChar.errorID := 16#0000_0000;
   instSequenceUnwinderCycle.instLConSMC_Winder.instTorquePrecontrol.instTableChar.y := 0.0;
   instSequenceUnwinderCycle.instLConSMC_Winder.instTorquePrecontrol.instTableChar.statEnableOld := FALSE;
   instSequenceUnwinderCycle.instLConSMC_Winder.instTorquePrecontrol.instTableChar.statLimitedSize := 0;
   instSequenceUnwinderCycle.instLConSMC_Winder.instTorquePrecontrol.instTableChar.statXval[0..20] := 0.0;
   instSequenceUnwinderCycle.instLConSMC_Winder.instTorquePrecontrol.instTableChar.statYval[0..20] := 0.0;
   instSequenceUnwinderCycle.instLConSMC_Winder.instTorquePrecontrol.instTableChar.statArrayCounter := 0;
   instSequenceUnwinderCycle.instLConSMC_Winder.instTorquePrecontrol.instTableChar.statMaxValueReached := FALSE;
   instSequenceUnwinderCycle.instLConSMC_Winder.instTorquePrecontrol.instTableChar.statReal1 := 0.0;
   instSequenceUnwinderCycle.instLConSMC_Winder.instTorquePrecontrol.instTableChar.statReal2 := 0.0;
   instSequenceUnwinderCycle.instLConSMC_Winder.instTorquePrecontrol.instTableChar.statReal3 := 0.0;
   instSequenceUnwinderCycle.instLConSMC_Winder.instTorquePrecontrol.instTableChar.statReal4 := 0.0;
   instSequenceUnwinderCycle.instLConSMC_Winder.instTorquePrecontrol.instTableChar.statFound := FALSE;
   instSequenceUnwinderCycle.instLConSMC_Winder.instTorquePrecontrol.instTableChar.statSegmentIndex := 0;
   instSequenceUnwinderCycle.instLConSMC_Winder.instTorquePrecontrol.instTableChar.statInt1 := 0;
   instSequenceUnwinderCycle.instLConSMC_Winder.instTorquePrecontrol.instTableChar.statEqualValues := FALSE;
   instSequenceUnwinderCycle.instLConSMC_Winder.instTorquePrecontrol.instTableChar.statError := FALSE;
   instSequenceUnwinderCycle.instLConSMC_Winder.instTorquePrecontrol.instTableChar.statBusy := FALSE;
   instSequenceUnwinderCycle.instLConSMC_Winder.instTorquePrecontrol.statAlpha := 0.0;
   instSequenceUnwinderCycle.instLConSMC_Winder.instTorquePrecontrol.statMfrict := 0.0;
   instSequenceUnwinderCycle.instLConSMC_Winder.instTorquePrecontrol.statMAccel := 0.0;
   instSequenceUnwinderCycle.instLConSMC_Winder.instTorquePrecontrol.statDiamActVal2 := 0.0;
   instSequenceUnwinderCycle.instLConSMC_Winder.instTorquePrecontrol.statDiamMin2 := 0.0;
   instSequenceUnwinderCycle.instLConSMC_Winder.instTorquePrecontrol.statDiamMax2 := 0.0;
   instSequenceUnwinderCycle.instLConSMC_Winder.instTorquePrecontrol.statGearRatio2 := 0.0;
   instSequenceUnwinderCycle.instLConSMC_Winder.instTorquePrecontrol.statWidth2 := 0.0;
   instSequenceUnwinderCycle.instLConSMC_Winder.instTorquePrecontrol.statSignWinderspeed := 0;
   instSequenceUnwinderCycle.instLConSMC_Winder.instTorquePrecontrol.statEnableold := FALSE;
   instSequenceUnwinderCycle.instLConSMC_Winder.instTorquePrecontrol.statBusy := FALSE;
   instSequenceUnwinderCycle.instLConSMC_Winder.instTorquePrecontrol.statMdDdt := 0.0;
   instSequenceUnwinderCycle.instLConSMC_Winder.instTorquePrecontrol.statDiamActOld := 0.0;
   instSequenceUnwinderCycle.instLConSMC_Winder.instTorquePrecontrol.statMConstRewinder := 0.0;
   instSequenceUnwinderCycle.instLConSMC_Winder.instLevelControl.run := FALSE;
   instSequenceUnwinderCycle.instLConSMC_Winder.instLevelControl.x := 0.0;
   instSequenceUnwinderCycle.instLConSMC_Winder.instLevelControl.alarmHigh := 100.0;
   instSequenceUnwinderCycle.instLConSMC_Winder.instLevelControl.warningHigh := 80.0;
   instSequenceUnwinderCycle.instLConSMC_Winder.instLevelControl.warningLow := -80.0;
   instSequenceUnwinderCycle.instLConSMC_Winder.instLevelControl.alarmLow := -100.0;
   instSequenceUnwinderCycle.instLConSMC_Winder.instLevelControl.hyst := 0.0;
   instSequenceUnwinderCycle.instLConSMC_Winder.instLevelControl.delayTime := T#3S;
   instSequenceUnwinderCycle.instLConSMC_Winder.instLevelControl.busy := FALSE;
   instSequenceUnwinderCycle.instLConSMC_Winder.instLevelControl.alarmUpperLimit := FALSE;
   instSequenceUnwinderCycle.instLConSMC_Winder.instLevelControl.alarmLowerLimit := FALSE;
   instSequenceUnwinderCycle.instLConSMC_Winder.instLevelControl.warningUpperLimit := FALSE;
   instSequenceUnwinderCycle.instLConSMC_Winder.instLevelControl.warningLowerLimit := FALSE;
   instSequenceUnwinderCycle.instLConSMC_Winder.instLevelControl.statAlarmUpperLimitSafe := FALSE;
   instSequenceUnwinderCycle.instLConSMC_Winder.instLevelControl.statWarningUpperLimitSafe := FALSE;
   instSequenceUnwinderCycle.instLConSMC_Winder.instLevelControl.statWarningLowerLimitSafe := FALSE;
   instSequenceUnwinderCycle.instLConSMC_Winder.instLevelControl.statAlarmLowerLimitSafe := FALSE;
   instSequenceUnwinderCycle.instLConSMC_Winder.instLevelControl.instTONalUp.PT := T#0MS;
   instSequenceUnwinderCycle.instLConSMC_Winder.instLevelControl.instTONalUp.IN := FALSE;
   instSequenceUnwinderCycle.instLConSMC_Winder.instLevelControl.instTONwaUp.PT := T#0MS;
   instSequenceUnwinderCycle.instLConSMC_Winder.instLevelControl.instTONwaUp.IN := FALSE;
   instSequenceUnwinderCycle.instLConSMC_Winder.instLevelControl.instTONwaLo.PT := T#0MS;
   instSequenceUnwinderCycle.instLConSMC_Winder.instLevelControl.instTONwaLo.IN := FALSE;
   instSequenceUnwinderCycle.instLConSMC_Winder.instLevelControl.instTONalLo.PT := T#0MS;
   instSequenceUnwinderCycle.instLConSMC_Winder.instLevelControl.instTONalLo.IN := FALSE;
   instSequenceUnwinderCycle.instLConSMC_Winder.instLevelControl.statAlarmUpperLimit := FALSE;
   instSequenceUnwinderCycle.instLConSMC_Winder.instLevelControl.statAlarmLowerLimit := FALSE;
   instSequenceUnwinderCycle.instLConSMC_Winder.instLevelControl.statWarningUpperLimit := FALSE;
   instSequenceUnwinderCycle.instLConSMC_Winder.instLevelControl.statWarningLowerLimit := FALSE;
   instSequenceUnwinderCycle.instLConSMC_Winder.instDiamCalc.enable := FALSE;
   instSequenceUnwinderCycle.instLConSMC_Winder.instDiamCalc.holdDiameter := FALSE;
   instSequenceUnwinderCycle.instLConSMC_Winder.instDiamCalc.metricUnits := TRUE;
   instSequenceUnwinderCycle.instLConSMC_Winder.instDiamCalc.setDiameter := FALSE;
   instSequenceUnwinderCycle.instLConSMC_Winder.instDiamCalc.lineFeedback := 0.0;
   instSequenceUnwinderCycle.instLConSMC_Winder.instDiamCalc.lineVelocity := 0.0;
   instSequenceUnwinderCycle.instLConSMC_Winder.instDiamCalc.windingShaftFeedback := 195.934;
   instSequenceUnwinderCycle.instLConSMC_Winder.instDiamCalc.shaftSpeed := 0.0;
   instSequenceUnwinderCycle.instLConSMC_Winder.instDiamCalc.selectDiamMode := 3;
   instSequenceUnwinderCycle.instLConSMC_Winder.instDiamCalc.typeOfWinder := 0;
   instSequenceUnwinderCycle.instLConSMC_Winder.instDiamCalc.tCycle := 10.0;
   instSequenceUnwinderCycle.instLConSMC_Winder.instDiamCalc.error := FALSE;
   instSequenceUnwinderCycle.instLConSMC_Winder.instDiamCalc.errorID := 16#0000_0000;
   instSequenceUnwinderCycle.instLConSMC_Winder.instDiamCalc.busy := FALSE;
   instSequenceUnwinderCycle.instLConSMC_Winder.instDiamCalc.diamModeInUse := 0;
   instSequenceUnwinderCycle.instLConSMC_Winder.instDiamCalc.atMinDia := FALSE;
   instSequenceUnwinderCycle.instLConSMC_Winder.instDiamCalc.atMaxDia := FALSE;
   instSequenceUnwinderCycle.instLConSMC_Winder.instDiamCalc.diamIsHold := FALSE;
   instSequenceUnwinderCycle.instLConSMC_Winder.instDiamCalc.calculatedWebThickness := 0.0;
   instSequenceUnwinderCycle.instLConSMC_Winder.instDiamCalc.diameter := 0.0;
   instSequenceUnwinderCycle.instLConSMC_Winder.instDiamCalc.statEnableOld := FALSE;
   instSequenceUnwinderCycle.instLConSMC_Winder.instDiamCalc.statBusy := FALSE;
   instSequenceUnwinderCycle.instLConSMC_Winder.instDiamCalc.statSetDiameter := FALSE;
   instSequenceUnwinderCycle.instLConSMC_Winder.instDiamCalc.statErrorLinePT1 := FALSE;
   instSequenceUnwinderCycle.instLConSMC_Winder.instDiamCalc.statErrorShaftPT1 := FALSE;
   instSequenceUnwinderCycle.instLConSMC_Winder.instDiamCalc.statErrorDiameterPT1 := FALSE;
   instSequenceUnwinderCycle.instLConSMC_Winder.instDiamCalc.statErrorLineInt := FALSE;
   instSequenceUnwinderCycle.instLConSMC_Winder.instDiamCalc.statDiamIsHold := FALSE;
   instSequenceUnwinderCycle.instLConSMC_Winder.instDiamCalc.statErrorShaftInt := FALSE;
   instSequenceUnwinderCycle.instLConSMC_Winder.instDiamCalc.statResetIntegrators := FALSE;
   instSequenceUnwinderCycle.instLConSMC_Winder.instDiamCalc.statDiamHoldImplicit := FALSE;
   instSequenceUnwinderCycle.instLConSMC_Winder.instDiamCalc.statCalculateFirstDiameter := FALSE;
   instSequenceUnwinderCycle.instLConSMC_Winder.instDiamCalc.statFirstDiameterOutputDone := FALSE;
   instSequenceUnwinderCycle.instLConSMC_Winder.instDiamCalc.statFirstDeltaEntered := FALSE;
   instSequenceUnwinderCycle.instLConSMC_Winder.instDiamCalc.statArrayEntryIntervalPassed := FALSE;
   instSequenceUnwinderCycle.instLConSMC_Winder.instDiamCalc.statOutputRateIntervalPassed := FALSE;
   instSequenceUnwinderCycle.instLConSMC_Winder.instDiamCalc.statLatchRawValue := FALSE;
   instSequenceUnwinderCycle.instLConSMC_Winder.instDiamCalc.statBufferFilled := FALSE;
   instSequenceUnwinderCycle.instLConSMC_Winder.instDiamCalc.statUseDactRawValue := FALSE;
   instSequenceUnwinderCycle.instLConSMC_Winder.instDiamCalc.statLatchNow := FALSE;
   instSequenceUnwinderCycle.instLConSMC_Winder.instDiamCalc.statSetDiameterValue := FALSE;
   instSequenceUnwinderCycle.instLConSMC_Winder.instDiamCalc.statWebThicknessNeeded := FALSE;
   instSequenceUnwinderCycle.instLConSMC_Winder.instDiamCalc.statPosBasedCalc := FALSE;
   instSequenceUnwinderCycle.instLConSMC_Winder.instDiamCalc.statDiamModeChanged := FALSE;
   instSequenceUnwinderCycle.instLConSMC_Winder.instDiamCalc.statInitializeDiamCalcPosition := FALSE;
   instSequenceUnwinderCycle.instLConSMC_Winder.instDiamCalc.statError := FALSE;
   instSequenceUnwinderCycle.instLConSMC_Winder.instDiamCalc.statErrorIDLinePT1 := 16#0000_0000;
   instSequenceUnwinderCycle.instLConSMC_Winder.instDiamCalc.statErrorIDShaftPT1 := 16#0000_0000;
   instSequenceUnwinderCycle.instLConSMC_Winder.instDiamCalc.statErrorIDDiameterPT1 := 16#0000_0000;
   instSequenceUnwinderCycle.instLConSMC_Winder.instDiamCalc.statErrorIDShaftInt := 16#0000_0000;
   instSequenceUnwinderCycle.instLConSMC_Winder.instDiamCalc.statErrorIDLineInt := 16#0000_0000;
   instSequenceUnwinderCycle.instLConSMC_Winder.instDiamCalc.statIntervalCounter := 0;
   instSequenceUnwinderCycle.instLConSMC_Winder.instDiamCalc.statDiamModeInUse := 0;
   instSequenceUnwinderCycle.instLConSMC_Winder.instDiamCalc.statArrayCounter := 0;
   instSequenceUnwinderCycle.instLConSMC_Winder.instDiamCalc.statRawDiameter := 0.0;
   instSequenceUnwinderCycle.instLConSMC_Winder.instDiamCalc.statDiameterInterpolated := 0.0;
   instSequenceUnwinderCycle.instLConSMC_Winder.instDiamCalc.statAbsLinVelocity := 0.0;
   instSequenceUnwinderCycle.instLConSMC_Winder.instDiamCalc.statAbsShaftSpeed := 0.0;
   instSequenceUnwinderCycle.instLConSMC_Winder.instDiamCalc.statCalcRoot := 0.0;
   instSequenceUnwinderCycle.instLConSMC_Winder.instDiamCalc.statRadiusOffset := 0.0;
   instSequenceUnwinderCycle.instLConSMC_Winder.instDiamCalc.statDiameterSetValLimited := 0.0;
   instSequenceUnwinderCycle.instLConSMC_Winder.instDiamCalc.statFirstArrayEntryPosition := 0.0;
   instSequenceUnwinderCycle.instLConSMC_Winder.instDiamCalc.statDeltaShaftRev := 0.0;
   instSequenceUnwinderCycle.instLConSMC_Winder.instDiamCalc.statDeltaLineRev := 0.0;
   instSequenceUnwinderCycle.instLConSMC_Winder.instDiamCalc.statDeltaShaft := 0.0;
   instSequenceUnwinderCycle.instLConSMC_Winder.instDiamCalc.statDeltaLine := 0.0;
   instSequenceUnwinderCycle.instLConSMC_Winder.instDiamCalc.statWindShaftStart := 0.0;
   instSequenceUnwinderCycle.instLConSMC_Winder.instDiamCalc.startLineStart := 0.0;
   instSequenceUnwinderCycle.instLConSMC_Winder.instDiamCalc.statBufferSize := 0.0;
   instSequenceUnwinderCycle.instLConSMC_Winder.instDiamCalc.statFloatingDeltaShaft := 0.0;
   instSequenceUnwinderCycle.instLConSMC_Winder.instDiamCalc.statFloatingDeltaLine := 0.0;
   instSequenceUnwinderCycle.instLConSMC_Winder.instDiamCalc.statDactRawValUnlimited := 0.0;
   instSequenceUnwinderCycle.instLConSMC_Winder.instDiamCalc.statWebThickness := 0.0;
   instSequenceUnwinderCycle.instLConSMC_Winder.instDiamCalc.statTargetDia := 0.0;
   instSequenceUnwinderCycle.instLConSMC_Winder.instDiamCalc.statTargetDiaLast := 0.0;
   instSequenceUnwinderCycle.instLConSMC_Winder.instDiamCalc.statTemp1 := 0.0;
   instSequenceUnwinderCycle.instLConSMC_Winder.instDiamCalc.statDeltaShaftArray[0..50] := 0.0;
   instSequenceUnwinderCycle.instLConSMC_Winder.instDiamCalc.statDeltaLineArray[0..50] := 0.0;
   instSequenceUnwinderCycle.instLConSMC_Winder.instDiamCalc.statDeltaArrayZero[0..50] := 0.0;
   instSequenceUnwinderCycle.instLConSMC_Winder.instDiamCalc.instLinePT1.set := FALSE;
   instSequenceUnwinderCycle.instLConSMC_Winder.instDiamCalc.instLinePT1.x := 0.0;
   instSequenceUnwinderCycle.instLConSMC_Winder.instDiamCalc.instLinePT1.setvalue := 0.0;
   instSequenceUnwinderCycle.instLConSMC_Winder.instDiamCalc.instLinePT1.smoothingTime := 100.0;
   instSequenceUnwinderCycle.instLConSMC_Winder.instDiamCalc.instLinePT1.tCycle := 0.0;
   instSequenceUnwinderCycle.instLConSMC_Winder.instDiamCalc.instLinePT1.error := FALSE;
   instSequenceUnwinderCycle.instLConSMC_Winder.instDiamCalc.instLinePT1.errorID := 16#0000_0000;
   instSequenceUnwinderCycle.instLConSMC_Winder.instDiamCalc.instLinePT1.y := 0.0;
   instSequenceUnwinderCycle.instLConSMC_Winder.instDiamCalc.instLinePT1.statTmax := 0.0;
   instSequenceUnwinderCycle.instLConSMC_Winder.instDiamCalc.instLinePT1.statXkm1 := 0.0;
   instSequenceUnwinderCycle.instLConSMC_Winder.instDiamCalc.instLinePT1.statYkm1 := 0.0;
   instSequenceUnwinderCycle.instLConSMC_Winder.instDiamCalc.instLinePT1.statFirstRun := TRUE;
   instSequenceUnwinderCycle.instLConSMC_Winder.instDiamCalc.instLinePT1.statY := 0.0;
   instSequenceUnwinderCycle.instLConSMC_Winder.instDiamCalc.instShaftPT1.set := FALSE;
   instSequenceUnwinderCycle.instLConSMC_Winder.instDiamCalc.instShaftPT1.x := 0.0;
   instSequenceUnwinderCycle.instLConSMC_Winder.instDiamCalc.instShaftPT1.setvalue := 0.0;
   instSequenceUnwinderCycle.instLConSMC_Winder.instDiamCalc.instShaftPT1.smoothingTime := 100.0;
   instSequenceUnwinderCycle.instLConSMC_Winder.instDiamCalc.instShaftPT1.tCycle := 0.0;
   instSequenceUnwinderCycle.instLConSMC_Winder.instDiamCalc.instShaftPT1.error := FALSE;
   instSequenceUnwinderCycle.instLConSMC_Winder.instDiamCalc.instShaftPT1.errorID := 16#0000_0000;
   instSequenceUnwinderCycle.instLConSMC_Winder.instDiamCalc.instShaftPT1.y := 0.0;
   instSequenceUnwinderCycle.instLConSMC_Winder.instDiamCalc.instShaftPT1.statTmax := 0.0;
   instSequenceUnwinderCycle.instLConSMC_Winder.instDiamCalc.instShaftPT1.statXkm1 := 0.0;
   instSequenceUnwinderCycle.instLConSMC_Winder.instDiamCalc.instShaftPT1.statYkm1 := 0.0;
   instSequenceUnwinderCycle.instLConSMC_Winder.instDiamCalc.instShaftPT1.statFirstRun := TRUE;
   instSequenceUnwinderCycle.instLConSMC_Winder.instDiamCalc.instShaftPT1.statY := 0.0;
   instSequenceUnwinderCycle.instLConSMC_Winder.instDiamCalc.instDiameterPT1.set := FALSE;
   instSequenceUnwinderCycle.instLConSMC_Winder.instDiamCalc.instDiameterPT1.x := 0.0;
   instSequenceUnwinderCycle.instLConSMC_Winder.instDiamCalc.instDiameterPT1.setvalue := 0.0;
   instSequenceUnwinderCycle.instLConSMC_Winder.instDiamCalc.instDiameterPT1.smoothingTime := 100.0;
   instSequenceUnwinderCycle.instLConSMC_Winder.instDiamCalc.instDiameterPT1.tCycle := 0.0;
   instSequenceUnwinderCycle.instLConSMC_Winder.instDiamCalc.instDiameterPT1.error := FALSE;
   instSequenceUnwinderCycle.instLConSMC_Winder.instDiamCalc.instDiameterPT1.errorID := 16#0000_0000;
   instSequenceUnwinderCycle.instLConSMC_Winder.instDiamCalc.instDiameterPT1.y := 0.0;
   instSequenceUnwinderCycle.instLConSMC_Winder.instDiamCalc.instDiameterPT1.statTmax := 0.0;
   instSequenceUnwinderCycle.instLConSMC_Winder.instDiamCalc.instDiameterPT1.statXkm1 := 0.0;
   instSequenceUnwinderCycle.instLConSMC_Winder.instDiamCalc.instDiameterPT1.statYkm1 := 0.0;
   instSequenceUnwinderCycle.instLConSMC_Winder.instDiamCalc.instDiameterPT1.statFirstRun := TRUE;
   instSequenceUnwinderCycle.instLConSMC_Winder.instDiamCalc.instDiameterPT1.statY := 0.0;
   instSequenceUnwinderCycle.instLConSMC_Winder.instDiamCalc.instShaftInt.set := FALSE;
   instSequenceUnwinderCycle.instLConSMC_Winder.instDiamCalc.instShaftInt.x := 0.0;
   instSequenceUnwinderCycle.instLConSMC_Winder.instDiamCalc.instShaftInt.setValue := 0.0;
   instSequenceUnwinderCycle.instLConSMC_Winder.instDiamCalc.instShaftInt.upperLimit := 1.0;
   instSequenceUnwinderCycle.instLConSMC_Winder.instDiamCalc.instShaftInt.lowerLimit := 0.0;
   instSequenceUnwinderCycle.instLConSMC_Winder.instDiamCalc.instShaftInt.integralTime := 5.0;
   instSequenceUnwinderCycle.instLConSMC_Winder.instDiamCalc.instShaftInt.tCycle := 0.0;
   instSequenceUnwinderCycle.instLConSMC_Winder.instDiamCalc.instShaftInt.error := FALSE;
   instSequenceUnwinderCycle.instLConSMC_Winder.instDiamCalc.instShaftInt.errorID := 16#0000_0000;
   instSequenceUnwinderCycle.instLConSMC_Winder.instDiamCalc.instShaftInt.upperLimitReached := FALSE;
   instSequenceUnwinderCycle.instLConSMC_Winder.instDiamCalc.instShaftInt.lowerLimitReached := FALSE;
   instSequenceUnwinderCycle.instLConSMC_Winder.instDiamCalc.instShaftInt.y := 0.0;
   instSequenceUnwinderCycle.instLConSMC_Winder.instDiamCalc.instShaftInt.statTmax := 0.0;
   instSequenceUnwinderCycle.instLConSMC_Winder.instDiamCalc.instShaftInt.statXkm1 := 0.0;
   instSequenceUnwinderCycle.instLConSMC_Winder.instDiamCalc.instShaftInt.statYkm1 := 0.0;
   instSequenceUnwinderCycle.instLConSMC_Winder.instDiamCalc.instShaftInt.statXFactor := 0.0;
   instSequenceUnwinderCycle.instLConSMC_Winder.instDiamCalc.instShaftInt.statFirstRun := TRUE;
   instSequenceUnwinderCycle.instLConSMC_Winder.instDiamCalc.instShaftInt.statUpperLimit := 0.0;
   instSequenceUnwinderCycle.instLConSMC_Winder.instDiamCalc.instShaftInt.statLowerLimit := 0.0;
   instSequenceUnwinderCycle.instLConSMC_Winder.instDiamCalc.instShaftInt.statLimiter := 0.0;
   instSequenceUnwinderCycle.instLConSMC_Winder.instDiamCalc.instShaftInt.statXlim := 0.0;
   instSequenceUnwinderCycle.instLConSMC_Winder.instDiamCalc.instShaftInt.statError := FALSE;
   instSequenceUnwinderCycle.instLConSMC_Winder.instDiamCalc.instShaftInt.statY := 0.0;
   instSequenceUnwinderCycle.instLConSMC_Winder.instDiamCalc.instLineInt.set := FALSE;
   instSequenceUnwinderCycle.instLConSMC_Winder.instDiamCalc.instLineInt.x := 0.0;
   instSequenceUnwinderCycle.instLConSMC_Winder.instDiamCalc.instLineInt.setValue := 0.0;
   instSequenceUnwinderCycle.instLConSMC_Winder.instDiamCalc.instLineInt.upperLimit := 1.0;
   instSequenceUnwinderCycle.instLConSMC_Winder.instDiamCalc.instLineInt.lowerLimit := 0.0;
   instSequenceUnwinderCycle.instLConSMC_Winder.instDiamCalc.instLineInt.integralTime := 5.0;
   instSequenceUnwinderCycle.instLConSMC_Winder.instDiamCalc.instLineInt.tCycle := 0.0;
   instSequenceUnwinderCycle.instLConSMC_Winder.instDiamCalc.instLineInt.error := FALSE;
   instSequenceUnwinderCycle.instLConSMC_Winder.instDiamCalc.instLineInt.errorID := 16#0000_0000;
   instSequenceUnwinderCycle.instLConSMC_Winder.instDiamCalc.instLineInt.upperLimitReached := FALSE;
   instSequenceUnwinderCycle.instLConSMC_Winder.instDiamCalc.instLineInt.lowerLimitReached := FALSE;
   instSequenceUnwinderCycle.instLConSMC_Winder.instDiamCalc.instLineInt.y := 0.0;
   instSequenceUnwinderCycle.instLConSMC_Winder.instDiamCalc.instLineInt.statTmax := 0.0;
   instSequenceUnwinderCycle.instLConSMC_Winder.instDiamCalc.instLineInt.statXkm1 := 0.0;
   instSequenceUnwinderCycle.instLConSMC_Winder.instDiamCalc.instLineInt.statYkm1 := 0.0;
   instSequenceUnwinderCycle.instLConSMC_Winder.instDiamCalc.instLineInt.statXFactor := 0.0;
   instSequenceUnwinderCycle.instLConSMC_Winder.instDiamCalc.instLineInt.statFirstRun := TRUE;
   instSequenceUnwinderCycle.instLConSMC_Winder.instDiamCalc.instLineInt.statUpperLimit := 0.0;
   instSequenceUnwinderCycle.instLConSMC_Winder.instDiamCalc.instLineInt.statLowerLimit := 0.0;
   instSequenceUnwinderCycle.instLConSMC_Winder.instDiamCalc.instLineInt.statLimiter := 0.0;
   instSequenceUnwinderCycle.instLConSMC_Winder.instDiamCalc.instLineInt.statXlim := 0.0;
   instSequenceUnwinderCycle.instLConSMC_Winder.instDiamCalc.instLineInt.statError := FALSE;
   instSequenceUnwinderCycle.instLConSMC_Winder.instDiamCalc.instLineInt.statY := 0.0;
   instSequenceUnwinderCycle.instLConSMC_Winder.instDiamCalc.instRTrigBusy.CLK := FALSE;
   instSequenceUnwinderCycle.instLConSMC_Winder.instDiamCalc.instRTrigBusy.Q := FALSE;
   instSequenceUnwinderCycle.instLConSMC_Winder.instDiamCalc.instRTrigBusy.Stat_Bit := FALSE;
   instSequenceUnwinderCycle.instLConSMC_Winder.instDiamCalc.instTrigArrayEntryIntervalPassed.CLK := FALSE;
   instSequenceUnwinderCycle.instLConSMC_Winder.instDiamCalc.instTrigArrayEntryIntervalPassed.Q := FALSE;
   instSequenceUnwinderCycle.instLConSMC_Winder.instDiamCalc.instTrigArrayEntryIntervalPassed.Stat_Bit := FALSE;
   instSequenceUnwinderCycle.instLConSMC_Winder.instDiamCalc.instTrigHold.CLK := FALSE;
   instSequenceUnwinderCycle.instLConSMC_Winder.instDiamCalc.instTrigHold.Q := FALSE;
   instSequenceUnwinderCycle.instLConSMC_Winder.instDiamCalc.instTrigHold.Stat_Bit := FALSE;
   instSequenceUnwinderCycle.instLConSMC_Winder.instDiamCalc.statSetDiameterOld := FALSE;
   instSequenceUnwinderCycle.instLConSMC_Winder.instIntAddVelo.set := TRUE;
   instSequenceUnwinderCycle.instLConSMC_Winder.instIntAddVelo.x := 0.0;
   instSequenceUnwinderCycle.instLConSMC_Winder.instIntAddVelo.setValue := 0.0;
   instSequenceUnwinderCycle.instLConSMC_Winder.instIntAddVelo.upperLimit := 1000000000000.0;
   instSequenceUnwinderCycle.instLConSMC_Winder.instIntAddVelo.lowerLimit := -1000000000000.0;
   instSequenceUnwinderCycle.instLConSMC_Winder.instIntAddVelo.integralTime := 1000.0;
   instSequenceUnwinderCycle.instLConSMC_Winder.instIntAddVelo.tCycle := 10.0;
   instSequenceUnwinderCycle.instLConSMC_Winder.instIntAddVelo.error := FALSE;
   instSequenceUnwinderCycle.instLConSMC_Winder.instIntAddVelo.errorID := 16#0000_0000;
   instSequenceUnwinderCycle.instLConSMC_Winder.instIntAddVelo.upperLimitReached := FALSE;
   instSequenceUnwinderCycle.instLConSMC_Winder.instIntAddVelo.lowerLimitReached := FALSE;
   instSequenceUnwinderCycle.instLConSMC_Winder.instIntAddVelo.y := 0.0;
   instSequenceUnwinderCycle.instLConSMC_Winder.instIntAddVelo.statTmax := 1000.0;
   instSequenceUnwinderCycle.instLConSMC_Winder.instIntAddVelo.statXkm1 := 0.0;
   instSequenceUnwinderCycle.instLConSMC_Winder.instIntAddVelo.statYkm1 := 0.0;
   instSequenceUnwinderCycle.instLConSMC_Winder.instIntAddVelo.statXFactor := 0.0;
   instSequenceUnwinderCycle.instLConSMC_Winder.instIntAddVelo.statFirstRun := FALSE;
   instSequenceUnwinderCycle.instLConSMC_Winder.instIntAddVelo.statUpperLimit := 1000000000000.0;
   instSequenceUnwinderCycle.instLConSMC_Winder.instIntAddVelo.statLowerLimit := -1000000000000.0;
   instSequenceUnwinderCycle.instLConSMC_Winder.instIntAddVelo.statLimiter := 0.0;
   instSequenceUnwinderCycle.instLConSMC_Winder.instIntAddVelo.statXlim := 0.0;
   instSequenceUnwinderCycle.instLConSMC_Winder.instIntAddVelo.statError := FALSE;
   instSequenceUnwinderCycle.instLConSMC_Winder.instIntAddVelo.statY := 0.0;
   instSequenceUnwinderCycle.instLConSMC_Winder.instMoveAvg.enable := FALSE;
   instSequenceUnwinderCycle.instLConSMC_Winder.instMoveAvg.updateConfig := FALSE;
   instSequenceUnwinderCycle.instLConSMC_Winder.instMoveAvg.sampleMode := 1;
   instSequenceUnwinderCycle.instLConSMC_Winder.instMoveAvg.inputSignal := 0.0;
   instSequenceUnwinderCycle.instLConSMC_Winder.instMoveAvg.subsetLength := 1;
   instSequenceUnwinderCycle.instLConSMC_Winder.instMoveAvg.samplingFactor := 1;
   instSequenceUnwinderCycle.instLConSMC_Winder.instMoveAvg.setTimePeriod := T#10MS;
   instSequenceUnwinderCycle.instLConSMC_Winder.instMoveAvg.cycleTime := 10000000;
   instSequenceUnwinderCycle.instLConSMC_Winder.instMoveAvg.error := FALSE;
   instSequenceUnwinderCycle.instLConSMC_Winder.instMoveAvg.errorID := 16#0000_0000;
   instSequenceUnwinderCycle.instLConSMC_Winder.instMoveAvg.samplingTime := 0.0;
   instSequenceUnwinderCycle.instLConSMC_Winder.instMoveAvg.timePeriod := 0.0;
   instSequenceUnwinderCycle.instLConSMC_Winder.instMoveAvg.shiftedInputSignal := 0.0;
   instSequenceUnwinderCycle.instLConSMC_Winder.instMoveAvg.movingAverage := 0.0;
   instSequenceUnwinderCycle.instLConSMC_Winder.instMoveAvg.statUpdateConfigOld := FALSE;
   instSequenceUnwinderCycle.instLConSMC_Winder.instMoveAvg.statEnableOld := FALSE;
   instSequenceUnwinderCycle.instLConSMC_Winder.instMoveAvg.statError := FALSE;
   instSequenceUnwinderCycle.instLConSMC_Winder.instMoveAvg.statSum := 0.0;
   instSequenceUnwinderCycle.instLConSMC_Winder.instMoveAvg.statSignalBufferSum[1..100] := 0.0;
   instSequenceUnwinderCycle.instLConSMC_Winder.instMoveAvg.statSamplingFactor := 1;
   instSequenceUnwinderCycle.instLConSMC_Winder.instMoveAvg.statSubsetLength := 1;
   instSequenceUnwinderCycle.instLConSMC_Winder.instMoveAvg.instfbUpdateConfig.fb_ID := 16#0426_0000;
   instSequenceUnwinderCycle.instLConSMC_Winder.instMoveAvg.instfbUpdateConfig.cascadeCalculation := FALSE;
   instSequenceUnwinderCycle.instLConSMC_Winder.instMoveAvg.instfbUpdateConfig.sampleMode := 1;
   instSequenceUnwinderCycle.instLConSMC_Winder.instMoveAvg.instfbUpdateConfig.maxBufferLengthMain := 100;
   instSequenceUnwinderCycle.instLConSMC_Winder.instMoveAvg.instfbUpdateConfig.maxBufferLengthSub := 10;
   instSequenceUnwinderCycle.instLConSMC_Winder.instMoveAvg.instfbUpdateConfig.inSubsetLengthMain := 1;
   instSequenceUnwinderCycle.instLConSMC_Winder.instMoveAvg.instfbUpdateConfig.setTimePeriod := T#10MS;
   instSequenceUnwinderCycle.instLConSMC_Winder.instMoveAvg.instfbUpdateConfig.inSamplingFactor := 1;
   instSequenceUnwinderCycle.instLConSMC_Winder.instMoveAvg.instfbUpdateConfig.cycleTime := 10000000;
   instSequenceUnwinderCycle.instLConSMC_Winder.instMoveAvg.instfbUpdateConfig.error := FALSE;
   instSequenceUnwinderCycle.instLConSMC_Winder.instMoveAvg.instfbUpdateConfig.errorID := 16#0000_0000;
   instSequenceUnwinderCycle.instLConSMC_Winder.instMoveAvg.instfbUpdateConfig.outSamplingFactorMain := 1;
   instSequenceUnwinderCycle.instLConSMC_Winder.instMoveAvg.instfbUpdateConfig.outSamplingFactorSub := 0;
   instSequenceUnwinderCycle.instLConSMC_Winder.instMoveAvg.instfbUpdateConfig.outSubsetLengthMain := 1;
   instSequenceUnwinderCycle.instLConSMC_Winder.instMoveAvg.instfbUpdateConfig.outSubsetLengthSub := 0;
   instSequenceUnwinderCycle.instLConSMC_Winder.instMoveAvg.instfbUpdateConfig.samplingTime := 10.0;
   instSequenceUnwinderCycle.instLConSMC_Winder.instMoveAvg.instfbUpdateConfig.actualizationRate := 0.0;
   instSequenceUnwinderCycle.instLConSMC_Winder.instMoveAvg.instfbUpdateConfig.timePeriod := 0.0;
   instSequenceUnwinderCycle.instLConSMC_Winder.instMoveAvg.instfbUpdateConfig.statError := FALSE;
   instSequenceUnwinderCycle.instLConSMC_Winder.instMoveAvg.instfbUpdateConfig.statErrorID := 16#0000_0000;
   instSequenceUnwinderCycle.instLConSMC_Winder.instMoveAvg.instfbUpdateConfig.statTimePeriodOut := 0.0;
   instSequenceUnwinderCycle.instLConSMC_Winder.instMoveAvg.instfbUpdateConfig.statActualizationRate := 0.0;
   instSequenceUnwinderCycle.instLConSMC_Winder.instMoveAvg.instfbUpdateConfig.statOutSamplingFactorSub := 0;
   instSequenceUnwinderCycle.instLConSMC_Winder.instMoveAvg.instfbUpdateConfig.statOutSubsetLengthSub := 0;
   instSequenceUnwinderCycle.instLConSMC_Winder.instMoveAvg.instfbUpdateConfig.statSamplingTime := 10.0;
   instSequenceUnwinderCycle.instLConSMC_Winder.instMoveAvg.instfbUpdateConfig.statOutSubsetLengthMain := 1;
   instSequenceUnwinderCycle.instLConSMC_Winder.instMoveAvg.instfbUpdateConfig.statOutSamplingFactorMain := 1;
   instSequenceUnwinderCycle.instLConSMC_Winder.instMoveAvg.instfbUpdateConfig.statCalcInMilliSecResol := FALSE;
   instSequenceUnwinderCycle.instLConSMC_Winder.instMoveAvg.instfbUpdateConfig.statCurrentSubLen := 0;
   instSequenceUnwinderCycle.instLConSMC_Winder.instMoveAvg.instfbUpdateConfig.statTimePeriod := 0;
   instSequenceUnwinderCycle.instLConSMC_Winder.instMoveAvg.instfbUpdateConfig.statDivisionRest := 0;
   instSequenceUnwinderCycle.instLConSMC_Winder.instMoveAvg.instfbUpdateConfig.statDivisionRestSub := 0;
   instSequenceUnwinderCycle.instLConSMC_Winder.instMoveAvg.instfbUpdateConfig.statRateToInteger := 0;
   instSequenceUnwinderCycle.instLConSMC_Winder.instMoveAvg.instfbUpdateConfig.statCycleTime := 10000;
   instSequenceUnwinderCycle.instLConSMC_Winder.instMoveAvg.instfbSumCalc.enable := FALSE;
   instSequenceUnwinderCycle.instLConSMC_Winder.instMoveAvg.instfbSumCalc.inputSignal := 0.0;
   instSequenceUnwinderCycle.instLConSMC_Winder.instMoveAvg.instfbSumCalc.inSubsetLength := 10;
   instSequenceUnwinderCycle.instLConSMC_Winder.instMoveAvg.instfbSumCalc.inRateOfSumCalc := 1;
   instSequenceUnwinderCycle.instLConSMC_Winder.instMoveAvg.instfbSumCalc.sumCalcUpdated := FALSE;
   instSequenceUnwinderCycle.instLConSMC_Winder.instMoveAvg.instfbSumCalc.sum := 0.0;
   instSequenceUnwinderCycle.instLConSMC_Winder.instMoveAvg.instfbSumCalc.shiftedInputSignal := 0.0;
   instSequenceUnwinderCycle.instLConSMC_Winder.instMoveAvg.instfbSumCalc.outSubsetLength := 10;
   instSequenceUnwinderCycle.instLConSMC_Winder.instMoveAvg.instfbSumCalc.statSumCalcUpdated := FALSE;
   instSequenceUnwinderCycle.instLConSMC_Winder.instMoveAvg.instfbSumCalc.statEnableOld := FALSE;
   instSequenceUnwinderCycle.instLConSMC_Winder.instMoveAvg.instfbSumCalc.statInitDone := FALSE;
   instSequenceUnwinderCycle.instLConSMC_Winder.instMoveAvg.instfbSumCalc.statIncreaseWindow := FALSE;
   instSequenceUnwinderCycle.instLConSMC_Winder.instMoveAvg.instfbSumCalc.statDecreaseWindow := FALSE;
   instSequenceUnwinderCycle.instLConSMC_Winder.instMoveAvg.instfbSumCalc.statEnableSumCalc := FALSE;
   instSequenceUnwinderCycle.instLConSMC_Winder.instMoveAvg.instfbSumCalc.statBufferPos := 1;
   instSequenceUnwinderCycle.instLConSMC_Winder.instMoveAvg.instfbSumCalc.statBufferPosResizeWindow := 0;
   instSequenceUnwinderCycle.instLConSMC_Winder.instMoveAvg.instfbSumCalc.statOldSubsetLength := 0;
   instSequenceUnwinderCycle.instLConSMC_Winder.instMoveAvg.instfbSumCalc.statChangedInSubsetLength := 10;
   instSequenceUnwinderCycle.instLConSMC_Winder.instMoveAvg.instfbSumCalc.statRateCounter := 1;
   instSequenceUnwinderCycle.instLConSMC_Winder.instMoveAvg.instfbSumCalc.statPosOfCenteredValue := 0;
   instSequenceUnwinderCycle.instLConSMC_Winder.instMoveAvg.instfbSumCalc.statOutSubsetLength := 0;
   instSequenceUnwinderCycle.instLConSMC_Winder.instMoveAvg.instfbSumCalc.statShiftedInputSignal := 0.0;
   instSequenceUnwinderCycle.instLConSMC_Winder.instMoveAvg.instfbSumCalc.statSum := 0.0;
   instSequenceUnwinderCycle.instLConSMC_Winder.instMoveAvg.statEnableRisingEdge := FALSE;
   instSequenceUnwinderCycle.instLConSMC_Winder.instMoveAvg.statCurrentSubLen := 0;
   instSequenceUnwinderCycle.instLConSMC_Winder.instSetAxisSTW.enable := FALSE;
   instSequenceUnwinderCycle.instLConSMC_Winder.instSetAxisSTW.resetSpeedInt := FALSE;
   instSequenceUnwinderCycle.instLConSMC_Winder.instSetAxisSTW.maskMotorBlockedFault := FALSE;
   instSequenceUnwinderCycle.instLConSMC_Winder.instSetAxisSTW.axis := 141;
   instSequenceUnwinderCycle.instLConSMC_Winder.instSetAxisSTW.integratorResetDone := FALSE;
   instSequenceUnwinderCycle.instLConSMC_Winder.instSetAxisSTW.maskMotorBlockedFaultDone := FALSE;
   instSequenceUnwinderCycle.instLConSMC_Winder.instSetAxisSTW.busy := FALSE;
   instSequenceUnwinderCycle.instLConSMC_Winder.instSetAxisSTW.error := FALSE;
   instSequenceUnwinderCycle.instLConSMC_Winder.instSetAxisSTW.errorID := 16#0000;
   instSequenceUnwinderCycle.instLConSMC_Winder.instSetAxisSTW.instSetAxisSTW.Execute := FALSE;
   instSequenceUnwinderCycle.instLConSMC_Winder.instSetAxisSTW.instSetAxisSTW.STW1 := 16#0000;
   instSequenceUnwinderCycle.instLConSMC_Winder.instSetAxisSTW.instSetAxisSTW.STW1BitMask := 16#0000;
   instSequenceUnwinderCycle.instLConSMC_Winder.instSetAxisSTW.instSetAxisSTW.STW2 := 16#0000;
   instSequenceUnwinderCycle.instLConSMC_Winder.instSetAxisSTW.instSetAxisSTW.STW2BitMask := 16#0000;
   instSequenceUnwinderCycle.instLConSMC_Winder.instSetAxisSTW.instSetAxisSTW.Done := FALSE;
   instSequenceUnwinderCycle.instLConSMC_Winder.instSetAxisSTW.instSetAxisSTW.Busy := FALSE;
   instSequenceUnwinderCycle.instLConSMC_Winder.instSetAxisSTW.instSetAxisSTW.CommandAborted := FALSE;
   instSequenceUnwinderCycle.instLConSMC_Winder.instSetAxisSTW.instSetAxisSTW.Error := FALSE;
   instSequenceUnwinderCycle.instLConSMC_Winder.instSetAxisSTW.instSetAxisSTW.ErrorId := 16#0000;
   instSequenceUnwinderCycle.instLConSMC_Winder.instSetAxisSTW.instRTrigResetIntegrator.CLK := FALSE;
   instSequenceUnwinderCycle.instLConSMC_Winder.instSetAxisSTW.instRTrigResetIntegrator.Q := FALSE;
   instSequenceUnwinderCycle.instLConSMC_Winder.instSetAxisSTW.instRTrigResetIntegrator.Stat_Bit := FALSE;
   instSequenceUnwinderCycle.instLConSMC_Winder.instSetAxisSTW.instRTrigMaskMotorBlockedFault.CLK := FALSE;
   instSequenceUnwinderCycle.instLConSMC_Winder.instSetAxisSTW.instRTrigMaskMotorBlockedFault.Q := FALSE;
   instSequenceUnwinderCycle.instLConSMC_Winder.instSetAxisSTW.instRTrigMaskMotorBlockedFault.Stat_Bit := FALSE;
   instSequenceUnwinderCycle.instLConSMC_Winder.instSetAxisSTW.instRTrigDisableActive.CLK := FALSE;
   instSequenceUnwinderCycle.instLConSMC_Winder.instSetAxisSTW.instRTrigDisableActive.Q := FALSE;
   instSequenceUnwinderCycle.instLConSMC_Winder.instSetAxisSTW.instRTrigDisableActive.Stat_Bit := FALSE;
   instSequenceUnwinderCycle.instLConSMC_Winder.instSetAxisSTW.instFTrigMaskMotorBlockedFault.CLK := FALSE;
   instSequenceUnwinderCycle.instLConSMC_Winder.instSetAxisSTW.instFTrigMaskMotorBlockedFault.Q := FALSE;
   instSequenceUnwinderCycle.instLConSMC_Winder.instSetAxisSTW.instFTrigMaskMotorBlockedFault.Stat_Bit := FALSE;
   instSequenceUnwinderCycle.instLConSMC_Winder.instSetAxisSTW.statEnableResetIntegrator := FALSE;
   instSequenceUnwinderCycle.instLConSMC_Winder.instSetAxisSTW.statEnableResetIntegratorOld := FALSE;
   instSequenceUnwinderCycle.instLConSMC_Winder.instSetAxisSTW.statDisableResetIntegrator := FALSE;
   instSequenceUnwinderCycle.instLConSMC_Winder.instSetAxisSTW.statResetIntegratorDone := FALSE;
   instSequenceUnwinderCycle.instLConSMC_Winder.instSetAxisSTW.statResetIntegratorDoneOld := FALSE;
   instSequenceUnwinderCycle.instLConSMC_Winder.instSetAxisSTW.statMaskMotorBlockedFaultActive := FALSE;
   instSequenceUnwinderCycle.instLConSMC_Winder.instSetAxisSTW.statEnableMaskMotorBlockedFault := FALSE;
   instSequenceUnwinderCycle.instLConSMC_Winder.instSetAxisSTW.statDisableMaskMotorBlockedFault := FALSE;
   instSequenceUnwinderCycle.instLConSMC_Winder.instSetAxisSTW.statBusy := FALSE;
   instSequenceUnwinderCycle.instLConSMC_Winder.instSetAxisSTW.statDisableActive := FALSE;
   instSequenceUnwinderCycle.instLConSMC_Winder.instSetAxisSTW.statEnableOld := FALSE;
   instSequenceUnwinderCycle.instLConSMC_Winder.instGetActualTension.enable := FALSE;
   instSequenceUnwinderCycle.instLConSMC_Winder.instGetActualTension.positiveTensionTorque := TRUE;
   instSequenceUnwinderCycle.instLConSMC_Winder.instGetActualTension.preCtrlMotor := 0.0;
   instSequenceUnwinderCycle.instLConSMC_Winder.instGetActualTension.diameter := 0.0;
   instSequenceUnwinderCycle.instLConSMC_Winder.instGetActualTension.actualTorque := 0.0;
   instSequenceUnwinderCycle.instLConSMC_Winder.instGetActualTension.gearRatio := 1.0;
   instSequenceUnwinderCycle.instLConSMC_Winder.instGetActualTension.valid := FALSE;
   instSequenceUnwinderCycle.instLConSMC_Winder.instGetActualTension.busy := FALSE;
   instSequenceUnwinderCycle.instLConSMC_Winder.instGetActualTension.error := FALSE;
   instSequenceUnwinderCycle.instLConSMC_Winder.instGetActualTension.status := 16#7000;
   instSequenceUnwinderCycle.instLConSMC_Winder.instGetActualTension.tensionActual := 0.0;
   instSequenceUnwinderCycle.instLConSMC_Winder.instGetActualTension.statEnableOld := FALSE;
   instSequenceUnwinderCycle.instLConSMC_Winder.instGetActualTension.statValid := FALSE;
   instSequenceUnwinderCycle.instLConSMC_Winder.instGetActualTension.statBusy := FALSE;
   instSequenceUnwinderCycle.instLConSMC_Winder.instGetActualTension.statError := FALSE;
   instSequenceUnwinderCycle.instLConSMC_Winder.instGetActualTension.statErrorUserCleared := FALSE;
   instSequenceUnwinderCycle.instLConSMC_Winder.instGetActualTension.statErrorAutoCleared := FALSE;
   instSequenceUnwinderCycle.instLConSMC_Winder.instGetActualTension.statStatus := 16#7000;
   instSequenceUnwinderCycle.instLConSMC_Winder.instGetActualTension.statFBState := 0;
   instSequenceUnwinderCycle.instLConSMC_Winder.instGetActualTension.statDisablingCompleted := FALSE;
   instSequenceUnwinderCycle.instLConSMC_Winder.instGetActualTension.statTensionActual := 0.0;
   instSequenceUnwinderCycle.instLConSMC_Winder.instGetActualTension.statTensionTorque := 0.0;
   instSequenceUnwinderCycle.instLConSMC_Winder.instOverspeedMonitoring.enable := FALSE;
   instSequenceUnwinderCycle.instLConSMC_Winder.instOverspeedMonitoring.reset := FALSE;
   instSequenceUnwinderCycle.instLConSMC_Winder.instOverspeedMonitoring.vLine := 0.0;
   instSequenceUnwinderCycle.instLConSMC_Winder.instOverspeedMonitoring.vOverride := 0.0;
   instSequenceUnwinderCycle.instLConSMC_Winder.instOverspeedMonitoring.vAct := 0.0;
   instSequenceUnwinderCycle.instLConSMC_Winder.instOverspeedMonitoring.velocityDeviationLimit := 20.0;
   instSequenceUnwinderCycle.instLConSMC_Winder.instOverspeedMonitoring.tCycle := 10.0;
   instSequenceUnwinderCycle.instLConSMC_Winder.instOverspeedMonitoring.valid := FALSE;
   instSequenceUnwinderCycle.instLConSMC_Winder.instOverspeedMonitoring.busy := FALSE;
   instSequenceUnwinderCycle.instLConSMC_Winder.instOverspeedMonitoring.error := FALSE;
   instSequenceUnwinderCycle.instLConSMC_Winder.instOverspeedMonitoring.status := 16#7000;
   instSequenceUnwinderCycle.instLConSMC_Winder.instOverspeedMonitoring.effectiveLimit := 0.0;
   instSequenceUnwinderCycle.instLConSMC_Winder.instOverspeedMonitoring.runAway := FALSE;
   instSequenceUnwinderCycle.instLConSMC_Winder.instOverspeedMonitoring.preControlAdjust := 1.0;
   instSequenceUnwinderCycle.instLConSMC_Winder.instOverspeedMonitoring.statEnableOld := FALSE;
   instSequenceUnwinderCycle.instLConSMC_Winder.instOverspeedMonitoring.statValid := FALSE;
   instSequenceUnwinderCycle.instLConSMC_Winder.instOverspeedMonitoring.statBusy := FALSE;
   instSequenceUnwinderCycle.instLConSMC_Winder.instOverspeedMonitoring.statError := FALSE;
   instSequenceUnwinderCycle.instLConSMC_Winder.instOverspeedMonitoring.statErrorUserCleared := FALSE;
   instSequenceUnwinderCycle.instLConSMC_Winder.instOverspeedMonitoring.statErrorAutoCleared := FALSE;
   instSequenceUnwinderCycle.instLConSMC_Winder.instOverspeedMonitoring.statStatus := 16#7000;
   instSequenceUnwinderCycle.instLConSMC_Winder.instOverspeedMonitoring.statFBState := 0;
   instSequenceUnwinderCycle.instLConSMC_Winder.instOverspeedMonitoring.statDisablingCompleted := FALSE;
   instSequenceUnwinderCycle.instLConSMC_Winder.instOverspeedMonitoring.statABSvDiff := 0.0;
   instSequenceUnwinderCycle.instLConSMC_Winder.instOverspeedMonitoring.statvDiffAdjustment := 0.0;
   instSequenceUnwinderCycle.instLConSMC_Winder.instOverspeedMonitoring.statPrecontrolAdjust := 1.0;
   instSequenceUnwinderCycle.instLConSMC_Winder.instOverspeedMonitoring.instPT1.set := FALSE;
   instSequenceUnwinderCycle.instLConSMC_Winder.instOverspeedMonitoring.instPT1.x := 0.0;
   instSequenceUnwinderCycle.instLConSMC_Winder.instOverspeedMonitoring.instPT1.setvalue := 0.0;
   instSequenceUnwinderCycle.instLConSMC_Winder.instOverspeedMonitoring.instPT1.smoothingTime := 100.0;
   instSequenceUnwinderCycle.instLConSMC_Winder.instOverspeedMonitoring.instPT1.tCycle := 0.0;
   instSequenceUnwinderCycle.instLConSMC_Winder.instOverspeedMonitoring.instPT1.error := FALSE;
   instSequenceUnwinderCycle.instLConSMC_Winder.instOverspeedMonitoring.instPT1.errorID := 16#0000_0000;
   instSequenceUnwinderCycle.instLConSMC_Winder.instOverspeedMonitoring.instPT1.y := 0.0;
   instSequenceUnwinderCycle.instLConSMC_Winder.instOverspeedMonitoring.instPT1.statTmax := 0.0;
   instSequenceUnwinderCycle.instLConSMC_Winder.instOverspeedMonitoring.instPT1.statXkm1 := 0.0;
   instSequenceUnwinderCycle.instLConSMC_Winder.instOverspeedMonitoring.instPT1.statYkm1 := 0.0;
   instSequenceUnwinderCycle.instLConSMC_Winder.instOverspeedMonitoring.instPT1.statFirstRun := TRUE;
   instSequenceUnwinderCycle.instLConSMC_Winder.instOverspeedMonitoring.instPT1.statY := 0.0;
   instSequenceUnwinderCycle.instLConSMC_Winder.instOverspeedMonitoring.statRunAwayDetected := FALSE;
   instSequenceUnwinderCycle.instLConSMC_Winder.instOverspeedMonitoring.statResetOld := FALSE;
   instSequenceUnwinderCycle.instLConSMC_LineUnitConversion.lengthUnitInput := 1013;
   instSequenceUnwinderCycle.instLConSMC_LineUnitConversion.velocityUnitInput := 1062;
   instSequenceUnwinderCycle.instLConSMC_LineUnitConversion.formatLength := 0.01;
   instSequenceUnwinderCycle.instLConSMC_LineUnitConversion.lengthConversionFactor := 0.001;
   instSequenceUnwinderCycle.instLConSMC_LineUnitConversion.velocityConversionFactor := 0.06;
   instSequenceUnwinderCycle.instLConSMC_LineUnitConversion.accelerationConversionFactor := 0.001;
END_DATA_BLOCK
